REGION Network 2: Call: Diagnostic Profinet Devices
   // For diagnose the whole profinet devices of this PLC
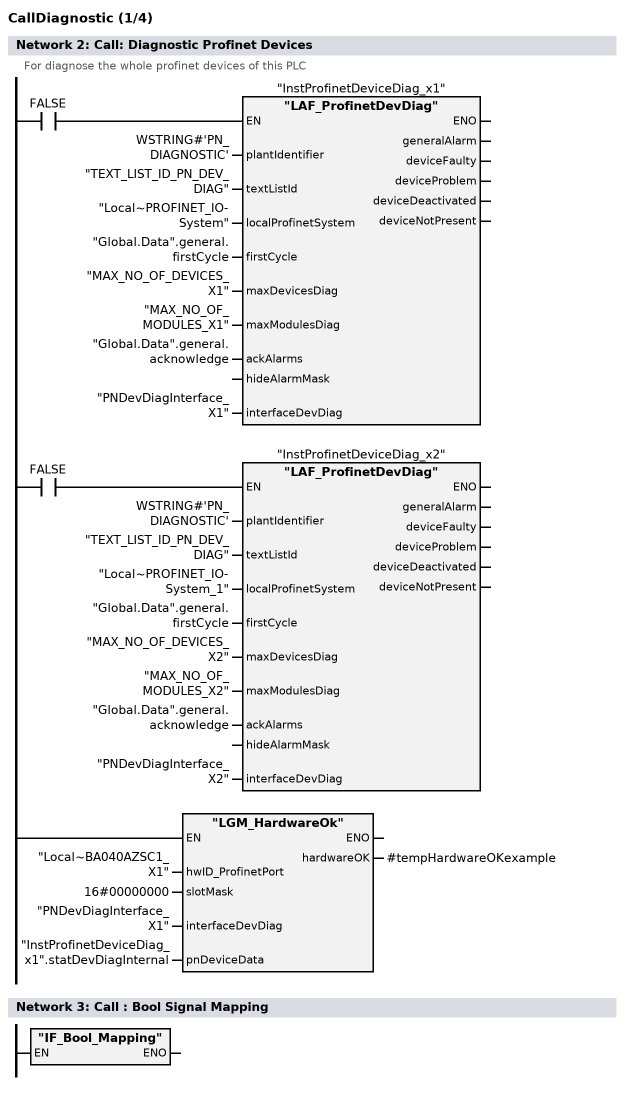
   RUNG wire#powerrail
      Contact( FALSE )
      "InstProfinetDeviceDiag_x1"(plantIdentifier := WSTRING#'PN_DIAGNOSTIC', textListId := "TEXT_LIST_ID_PN_DEV_DIAG", localProfinetSystem := "Local~PROFINET_IO-System", firstCycle := "Global.Data".general.firstCycle, maxDevicesDiag := "MAX_NO_OF_DEVICES_X1", maxModulesDiag := "MAX_NO_OF_MODULES_X1", ackAlarms := "Global.Data".general.acknowledge, hideAlarmMask :=, interfaceDevDiag := "PNDevDiagInterface_X1", generalAlarm =>, deviceFaulty =>, deviceProblem =>, deviceDeactivated =>, deviceNotPresent =>)
   END_RUNG
   RUNG wire#powerrail
      Contact( FALSE )
      "InstProfinetDeviceDiag_x2"(plantIdentifier := WSTRING#'PN_DIAGNOSTIC', textListId := "TEXT_LIST_ID_PN_DEV_DIAG", localProfinetSystem := "Local~PROFINET_IO-System_1", firstCycle := "Global.Data".general.firstCycle, maxDevicesDiag := "MAX_NO_OF_DEVICES_X2", maxModulesDiag := "MAX_NO_OF_MODULES_X2", ackAlarms := "Global.Data".general.acknowledge, hideAlarmMask :=, interfaceDevDiag := "PNDevDiagInterface_X2", generalAlarm =>, deviceFaulty =>, deviceProblem =>, deviceDeactivated =>, deviceNotPresent =>)
   END_RUNG
   RUNG wire#powerrail
      "LGM_HardwareOk"(hwID_ProfinetPort := "Local~BA040AZSC1_X1", slotMask := 16#00000000, interfaceDevDiag := "PNDevDiagInterface_X1", pnDeviceData := "InstProfinetDeviceDiag_x1".statDevDiagInternal, hardwareOK => #tempHardwareOKexample)
   END_RUNG
   // the same network as SCL:
   IF FALSE THEN
       "InstProfinetDeviceDiag_x1"(plantIdentifier := WSTRING#'PN_DIAGNOSTIC',   // "LAF_ProfinetDevDiag"
                               textListId := "TEXT_LIST_ID_PN_DEV_DIAG",
                               localProfinetSystem := "Local~PROFINET_IO-System",
                               firstCycle := "Global.Data".general.firstCycle,
                               maxDevicesDiag := "MAX_NO_OF_DEVICES_X1",
                               maxModulesDiag := "MAX_NO_OF_MODULES_X1",
                               ackAlarms := "Global.Data".general.acknowledge,
                               interfaceDevDiag := "PNDevDiagInterface_X1");
       "InstProfinetDeviceDiag_x2"(plantIdentifier := WSTRING#'PN_DIAGNOSTIC',   // "LAF_ProfinetDevDiag"
                               textListId := "TEXT_LIST_ID_PN_DEV_DIAG",
                               localProfinetSystem := "Local~PROFINET_IO-System_1",
                               firstCycle := "Global.Data".general.firstCycle,
                               maxDevicesDiag := "MAX_NO_OF_DEVICES_X2",
                               maxModulesDiag := "MAX_NO_OF_MODULES_X2",
                               ackAlarms := "Global.Data".general.acknowledge,
                               interfaceDevDiag := "PNDevDiagInterface_X2");
   END_IF;
   "LGM_HardwareOk"(hwID_ProfinetPort := "Local~BA040AZSC1_X1",
                    slotMask := 16#00000000,
                    interfaceDevDiag := "PNDevDiagInterface_X1",
                    pnDeviceData := "InstProfinetDeviceDiag_x1".statDevDiagInternal,
                    hardwareOK => #tempHardwareOKexample);
END_REGION

REGION Network 3: Call : Bool Signal Mapping
   RUNG wire#powerrail
      "IF_Bool_Mapping"()
   END_RUNG
   // the same network as SCL:
   "IF_Bool_Mapping"();
END_REGION

REGION Network 4: Call: Diagnostic Bool Interface Signals
   // Call the interface bool blocks to show boolean signals on the HMI
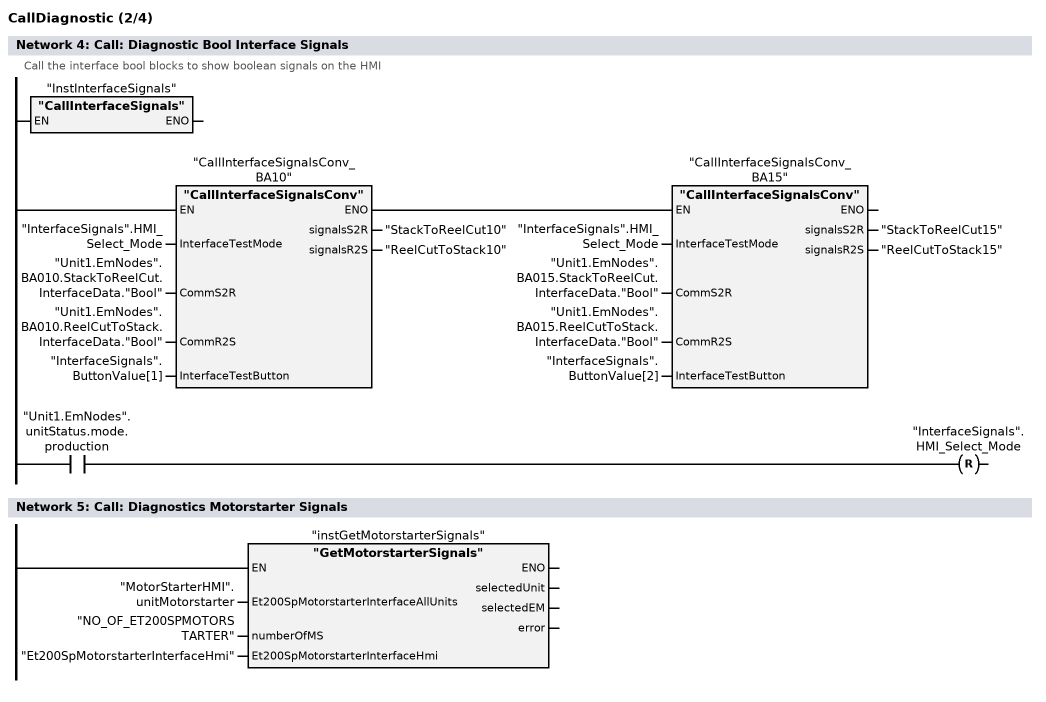
   RUNG wire#powerrail
      "InstInterfaceSignals"()
   END_RUNG
   RUNG wire#powerrail
      "CallInterfaceSignalsConv_BA10"(InterfaceTestMode := "InterfaceSignals".HMI_Select_Mode, CommS2R := "Unit1.EmNodes".BA010.StackToReelCut.InterfaceData."Bool", CommR2S := "Unit1.EmNodes".BA010.ReelCutToStack.InterfaceData."Bool", InterfaceTestButton := "InterfaceSignals".ButtonValue[1], signalsS2R => "StackToReelCut10", signalsR2S => "ReelCutToStack10")
      "CallInterfaceSignalsConv_BA15"(InterfaceTestMode := "InterfaceSignals".HMI_Select_Mode, CommS2R := "Unit1.EmNodes".BA015.StackToReelCut.InterfaceData."Bool", CommR2S := "Unit1.EmNodes".BA015.ReelCutToStack.InterfaceData."Bool", InterfaceTestButton := "InterfaceSignals".ButtonValue[2], signalsS2R => "StackToReelCut15", signalsR2S => "ReelCutToStack15")
   END_RUNG
   RUNG wire#powerrail
      Contact( "Unit1.EmNodes".unitStatus.mode.production )
      R_Coil( "InterfaceSignals".HMI_Select_Mode )
   END_RUNG
   // the same network as SCL:
   "InstInterfaceSignals"();   // "CallInterfaceSignals"
   "CallInterfaceSignalsConv_BA10"(InterfaceTestMode := "InterfaceSignals".HMI_Select_Mode,   // "CallInterfaceSignalsConv"
                           CommS2R := "Unit1.EmNodes".BA010.StackToReelCut.InterfaceData."Bool",
                           CommR2S := "Unit1.EmNodes".BA010.ReelCutToStack.InterfaceData."Bool",
                           InterfaceTestButton := "InterfaceSignals".ButtonValue[1],
                           signalsS2R => "StackToReelCut10",
                           signalsR2S => "ReelCutToStack10",
                           ENO => #_w1);
   IF #_w1 THEN
       "CallInterfaceSignalsConv_BA15"(InterfaceTestMode := "InterfaceSignals".HMI_Select_Mode,   // "CallInterfaceSignalsConv"
                               CommS2R := "Unit1.EmNodes".BA015.StackToReelCut.InterfaceData."Bool",
                               CommR2S := "Unit1.EmNodes".BA015.ReelCutToStack.InterfaceData."Bool",
                               InterfaceTestButton := "InterfaceSignals".ButtonValue[2],
                               signalsS2R => "StackToReelCut15",
                               signalsR2S => "ReelCutToStack15");
   END_IF;
   IF "Unit1.EmNodes".unitStatus.mode.production THEN "InterfaceSignals".HMI_Select_Mode := FALSE; END_IF;
END_REGION

REGION Network 5: Call: Diagnostics Motorstarter Signals
   RUNG wire#powerrail
      "instGetMotorstarterSignals"(Et200SpMotorstarterInterfaceAllUnits := "MotorStarterHMI".unitMotorstarter, numberOfMS := "NO_OF_ET200SPMOTORSTARTER", Et200SpMotorstarterInterfaceHmi := "Et200SpMotorstarterInterfaceHmi", selectedUnit =>, selectedEM =>, error =>)
   END_RUNG
   // the same network as SCL:
   "instGetMotorstarterSignals"(Et200SpMotorstarterInterfaceAllUnits := "MotorStarterHMI".unitMotorstarter,   // "GetMotorstarterSignals"
                           numberOfMS := "NO_OF_ET200SPMOTORSTARTER",
                           Et200SpMotorstarterInterfaceHmi := "Et200SpMotorstarterInterfaceHmi");
END_REGION

REGION Network 6: Call: Diagnostics Drives
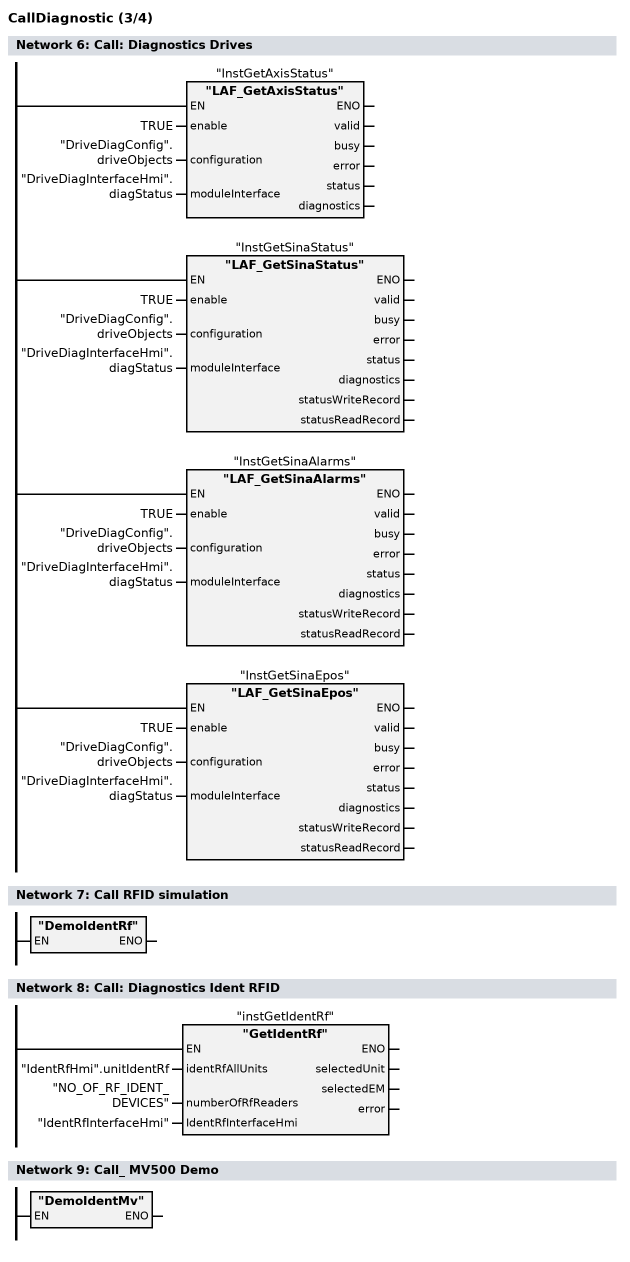
   RUNG wire#powerrail
      "InstGetAxisStatus"(enable := TRUE, configuration := "DriveDiagConfig".driveObjects, moduleInterface := "DriveDiagInterfaceHmi".diagStatus, valid =>, busy =>, error =>, status =>, diagnostics =>)
   END_RUNG
   RUNG wire#powerrail
      "InstGetSinaStatus"(enable := TRUE, configuration := "DriveDiagConfig".driveObjects, moduleInterface := "DriveDiagInterfaceHmi".diagStatus, valid =>, busy =>, error =>, status =>, diagnostics =>, statusWriteRecord =>, statusReadRecord =>)
   END_RUNG
   RUNG wire#powerrail
      "InstGetSinaAlarms"(enable := TRUE, configuration := "DriveDiagConfig".driveObjects, moduleInterface := "DriveDiagInterfaceHmi".diagStatus, valid =>, busy =>, error =>, status =>, diagnostics =>, statusWriteRecord =>, statusReadRecord =>)
   END_RUNG
   RUNG wire#powerrail
      "InstGetSinaEpos"(enable := TRUE, configuration := "DriveDiagConfig".driveObjects, moduleInterface := "DriveDiagInterfaceHmi".diagStatus, valid =>, busy =>, error =>, status =>, diagnostics =>, statusWriteRecord =>, statusReadRecord =>)
   END_RUNG
   // the same network as SCL:
   "InstGetAxisStatus"(enable := TRUE,   // "LAF_GetAxisStatus"
                       configuration := "DriveDiagConfig".driveObjects,
                       moduleInterface := "DriveDiagInterfaceHmi".diagStatus);
   "InstGetSinaStatus"(enable := TRUE,   // "LAF_GetSinaStatus"
                       configuration := "DriveDiagConfig".driveObjects,
                       moduleInterface := "DriveDiagInterfaceHmi".diagStatus);
   "InstGetSinaAlarms"(enable := TRUE,   // "LAF_GetSinaAlarms"
                       configuration := "DriveDiagConfig".driveObjects,
                       moduleInterface := "DriveDiagInterfaceHmi".diagStatus);
   "InstGetSinaEpos"(enable := TRUE,   // "LAF_GetSinaEpos"
                     configuration := "DriveDiagConfig".driveObjects,
                     moduleInterface := "DriveDiagInterfaceHmi".diagStatus);
END_REGION

REGION Network 7: Call RFID simulation
   RUNG wire#powerrail
      "DemoIdentRf"()
   END_RUNG
   // the same network as SCL:
   "DemoIdentRf"();
END_REGION

REGION Network 8: Call: Diagnostics Ident RFID
   RUNG wire#powerrail
      "instGetIdentRf"(identRfAllUnits := "IdentRfHmi".unitIdentRf, numberOfRfReaders := "NO_OF_RF_IDENT_DEVICES", IdentRfInterfaceHmi := "IdentRfInterfaceHmi", selectedUnit =>, selectedEM =>, error =>)
   END_RUNG
   // the same network as SCL:
   "instGetIdentRf"(identRfAllUnits := "IdentRfHmi".unitIdentRf,   // "GetIdentRf"
                    numberOfRfReaders := "NO_OF_RF_IDENT_DEVICES",
                    IdentRfInterfaceHmi := "IdentRfInterfaceHmi");
END_REGION

REGION Network 9: Call_ MV500 Demo
   RUNG wire#powerrail
      "DemoIdentMv"()
   END_RUNG
   // the same network as SCL:
   "DemoIdentMv"();
END_REGION

REGION Network 10: Call: Diagnosticsa Ident MV
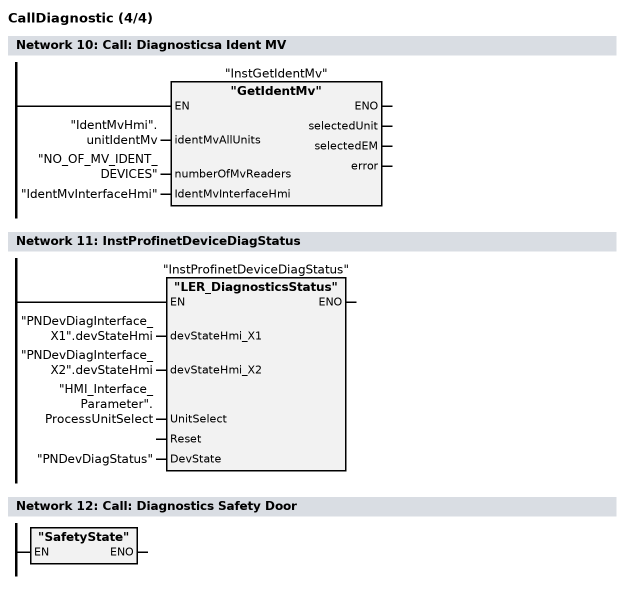
   RUNG wire#powerrail
      "InstGetIdentMv"(identMvAllUnits := "IdentMvHmi".unitIdentMv, numberOfMvReaders := "NO_OF_MV_IDENT_DEVICES", IdentMvInterfaceHmi := "IdentMvInterfaceHmi", selectedUnit =>, selectedEM =>, error =>)
   END_RUNG
   // the same network as SCL:
   "InstGetIdentMv"(identMvAllUnits := "IdentMvHmi".unitIdentMv,   // "GetIdentMv"
                    numberOfMvReaders := "NO_OF_MV_IDENT_DEVICES",
                    IdentMvInterfaceHmi := "IdentMvInterfaceHmi");
END_REGION

REGION Network 11: InstProfinetDeviceDiagStatus
   RUNG wire#powerrail
      "InstProfinetDeviceDiagStatus"(devStateHmi_X1 := "PNDevDiagInterface_X1".devStateHmi, devStateHmi_X2 := "PNDevDiagInterface_X2".devStateHmi, UnitSelect := "HMI_Interface_Parameter".ProcessUnitSelect, Reset :=, DevState := "PNDevDiagStatus")
   END_RUNG
   // the same network as SCL:
   "InstProfinetDeviceDiagStatus"(devStateHmi_X1 := "PNDevDiagInterface_X1".devStateHmi,   // "LER_DiagnosticsStatus"
                           devStateHmi_X2 := "PNDevDiagInterface_X2".devStateHmi,
                           UnitSelect := "HMI_Interface_Parameter".ProcessUnitSelect,
                           DevState := "PNDevDiagStatus");
END_REGION

REGION Network 12: Call: Diagnostics Safety Door
   RUNG wire#powerrail
      "SafetyState"()
   END_RUNG
   // the same network as SCL:
   "SafetyState"();
END_REGION
END_FUNCTION

FUNCTION "IF_Bool_Mapping" : Void
{ S7_Optimized_Access := 'TRUE' ; Published := 'FALSE' }
VERSION : 0.1

BEGIN
	// IO Mapping 25.12.10
	REGION BK
	    REGION BK01
	        "BK01"."X10-1.BTM DIRECTION CHECK SENSOR" := "BA040AZSBK01.00";
	        //"BK01"."X11-1.SPARE" := "BA030AZSBK01.I01";
	        //"BK01"."X12-1.SPARE" := "BA030AZSBK01.I02";
	        "BK01"."X13-1.COMPENSATOR #1 LIMIT SENSOR(-)" := "Sensor".EM3[0];
	        "BK01"."X14-1.COMPENSATOR #1 LIMIT SENSOR(+)" := "Sensor".EM3[1];
	        //"BK01"."X15-1.SPARE" := "BA030AZSBK01.I05";
	        //"BK01"."X16-1.SPARE" := "BA030AZSBK01.I06";
	        "BK01"."X17-1.SAFETY PIN IDLE POSITION" := "BA040AZSBK01.07";
	        "BK01"."X10-2.TOP DIRECTION CHECK SENSOR" := "BA040AZSBK01.10";
	        //"BK01"."X11-2.SPARE" := "BA030AZSBK01.I09";
	        //"BK01"."X12-2.SPARE" := "BA030AZSBK01.I10";
	        "BK01"."X13-2.COMPENSATOR #1 HOME SENSOR" := "Sensor".EM3[2];
	        //"BK01"."X14-2.SPARE" := "BA030AZSBK01.I12";
	        //"BK01"."X15-2.SPARE" := "BA030AZSBK01.I13";
	        //"BK01"."X16-2.SPARE" := "BA030AZSBK01.I14";
	        //"BK01"."X17-2.SPARE" := "BA030AZSBK01.I15";
	    END_REGION
	    REGION BK02
	        "BK02"."X10-1.SUCTION PAD TOP DOWN" := "BA040AZSBK02.00";
	        "BK02"."X11-1.SUCTION PAD BTM DOWN" := "BA040AZSBK02.01";
	        "BK02"."X12-1.CUTTER DOWN" := "BA040AZSBK02.02";
	        "BK02"."X13-1.TAPE TOP DOWN" := "BA040AZSBK02.03";
	        "BK02"."X14-1.TAPE BTM DOWN" := "BA040AZSBK02.04";
	        "BK02"."X15-1.SPLICE HEAD ROTATE TOP BACKWARD" := "BA040AZSBK02.05";
	        "BK02"."X16-1.SPLICE HEAD ROTATE BTM BACKWARD" := "BA040AZSBK02.06";
	        //"BK02"."X17-1.SPARE" := "BA030AZSBK02.I07";
	        "BK02"."X10-2.SUCTION PAD TOP UP" := "BA040AZSBK02.10";
	        "BK02"."X11-2.SUCTION PAD BTM UP" := "BA040AZSBK02.11";
	        "BK02"."X12-2.CUTTER UP" := "BA040AZSBK02.12";
	        "BK02"."X13-2.TAPE TOP UP" := "BA040AZSBK02.13";
	        "BK02"."X14-2.TAPE BTM UP" := "BA040AZSBK02.14";
	        "BK02"."X15-2.SPLICE HEAD ROTATE TOP FORWARD" := "BA040AZSBK02.15";
	        "BK02"."X16-2.SPLICE HEAD ROTATE BTM FORWARD" := "BA040AZSBK02.16";
	        //"BK02"."X17-2.SPARE" := "BA030AZSBK02.I15";
	    END_REGION
	    REGION BK03
	        "BK03"."X10-1.SUCTION PAD TOP LEFT PRESSURE SWITCH" := "BA040AZSBK03.00";
	        "BK03"."X10-2.SUCTION PAD TOP RIGHT PRESSURE SWITCH" := "BA040AZSBK03.01";
	        "BK03"."X12-1.SUCTION PAD BTM LEFT PRESSURE SWITCH" := "BA040AZSBK03.02";
	        "BK03"."X12-2.SUCTION PAD BTM RIGHT PRESSURE SWITCH" := "BA040AZSBK03.03";
	        "BK03"."X14-1.SUCTION PAD TOP TAPE PRESSURE SWITCH" := "BA040AZSBK03.04";
	        "BK03"."X14-2.SUCTION PAD BTM TAPE PRESSURE SWITCH" := "BA040AZSBK03.05";
	        "BK03"."X14-2.SUCTION PAD BTM TAPE PRESSURE SWITCH" := "BA040AZSBK03.06";
	        //"BK03"."X16-2.SPARE" := "BA030AZSBK03.I07";
	    END_REGION
	    REGION BK04
	        "BK04"."X10-1.CATHODE MAIN P&P1 LIMITS SENSOR(-)" := "Sensor".EM5[18];
	        "BK04"."X11-1.CATHODE MAIN P&P1 LIMITS SENSOR(+)" := "Sensor".EM5[19];
	        "BK04"."X12-1.CATHODE MAIN P&P2 LIMITS SENSOR(-)" := "Sensor".EM5[21];
	        "BK04"."X13-1.CATHODE MAIN P&P2 LIMITS SENSOR(+)" := "Sensor".EM5[22];
	        "BK04"."X14-1.ANODE MAIN P&P2 LIMITS SENSOR(-)" := "Sensor".EM4[0];
	        "BK04"."X15-1.ANODE MAIN P&P2 LIMITS SENSOR(+)" := "Sensor".EM4[1];
	        "BK04"."X16-1.ANODE MAIN P&P1 LIMITS SENSOR(-)" := "Sensor".EM4[21];
	        "BK04"."X17-1.ANODE MAIN P&P1 LIMITS SENSOR(+)" := "Sensor".EM4[22];
	        "BK04"."X10-2.CATHODE MAIN P&P1 LIMITS SENSOR HOME" := "Sensor".EM5[20];
	        //"BK04"."X11-2.SPARE" := "BA030AZSBK04.I09";
	        "BK04"."X12-2.CATHODE MAIN P&P2 LIMITS SENSOR HOME" := "Sensor".EM5[23];
	        //"BK04"."X13-2.SPARE" := "BA030AZSBK04.I11";
	        "BK04"."X14-2.ANODE MAIN P&P2 LIMITS SENSOR HOME" := "Sensor".EM4[2];
	        //"BK04"."X15-2.SPARE" := "BA030AZSBK04.I13";
	        "BK04"."X16-2.ANODE MAIN P&P1 LIMITS SENSOR HOME" := "Sensor".EM4[23];
	        //"BK04"."X17-2.SPARE" := "BA030AZSBK04.I15";
	    END_REGION
	    REGION BK05
	        "BK05"."X10-1.ANODE MAIN P&P1 Z-AXIS LIMIT SENSOR(-)" := "Sensor".EM4[3];
	        "BK05"."X11-1.ANODE MAIN P&P1 Z-AXIS LIMIT SENSOR(+)" := "Sensor".EM4[4];
	        "BK05"."X12-1.ANODE MAIN P&P1 Y-AXIS LIMIT SENSOR(-)" := "Sensor".EM4[5];
	        "BK05"."X13-1.ANODE MAIN P&P1 Y-AXIS LIMIT SENSOR(+)" := "Sensor".EM4[6];
	        //"BK05"."X14-1.SPARE" := "BA030AZSBK05.I04";
	        "BK05"."X15-1.ANODE MAIN P&P1 DETECT SENSOR" := "BA040AZSBK05.05";
	        "BK05"."X16-1.ANODE MAIN P&P1 ROTARY CCW" := "BA040AZSBK05.06";
	        "BK05"."X17-1.ANODE MAIN P&P1 PRESSURE SWITCH" := "BA040AZSBK05.07";
	        "BK05"."X10-2.ANODE MAIN P&P1 Z-AXIS HOME SENSOR" := "Sensor".EM4[7];
	        //"BK05"."X11-2.SPARE" := "BA030AZSBK05.I09";
	        "BK05"."X12-2.ANODE MAIN P&P1 Y-AXIS HOME SENSOR" := "Sensor".EM4[8];
	        //"BK05"."X13-2.SPARE" := "BA030AZSBK05.I11";
	        //"BK05"."X14-2.SPARE" := "BA030AZSBK05.I12";
	        //"BK05"."X15-2.SPARE" := "BA030AZSBK05.I13";
	        "BK05"."X16-2.ANODE MAIN P&P1 ROTARY CW" := "BA040AZSBK05.16";
	        //"BK05"."X17-2.SPARE" := "BA030AZSBK05.I15";
	    END_REGION BK06
	        "BK06"."X10-1.ANODE MAIN P&P2 Z-AXIS LIMIT SENSOR(-)" := "Sensor".EM4[9];
	        "BK06"."X10-2.ANODE MAIN P&P2 Z-AXIS HOME SENSOR" := "Sensor".EM4[10];
	        "BK06"."X12-1.ANODE MAIN P&P2 Z-AXIS LIMIT SENSOR(+)" := "Sensor".EM4[11];
	        "BK06"."X12-2.ANODE MAIN P&P2 DETECT SENSOR" := "BA040AZSBK06.03";
	        "BK06"."X14-1.ANODE MAIN P&P2 PRESSURE SWITCH" := "BA040AZSBK06.04";
	        //"BK06"."X14-2.SPARE" := "BA030AZSBK06.I05";
	        //"BK06"."X16-1.SPARE" := "BA030AZSBK06.I06";
	        //"BK06"."X16-2.SPARE" := "BA030AZSBK06.I07";
	    REGION BK07
	        "BK07"."X10-1.CATHODE MAIN P&P1 Z-AXIS LIMIT SENSOR(-)" := "Sensor".EM5[0];
	        "BK07"."X11-1.CATHODE MAIN P&P1 Z-AXIS LIMIT SENSOR(+)" := "Sensor".EM5[1];
	        "BK07"."X12-1.CATHODE MAIN P&P1 Y-AXIS LIMIT SENSOR(-)" := "Sensor".EM5[2];
	        "BK07"."X13-1.CATHODE MAIN P&P1 Y-AXIS LIMIT SENSOR(+)" := "Sensor".EM5[3];
	        //"BK07"."X14-1.SPARE" := "BA030AZSBK07.I04";
	        "BK07"."X15-1.CATHODE MAIN P&P1 DETECT SENSOR" := "BA040AZSBK07.05";
	        "BK07"."X16-1.CATHODE MAIN P&P1 ROTARY CCW" := "BA040AZSBK07.06";
	        "BK07"."X17-1.CATHODE MAIN P&P1 PRESSURE SWITCH" := "BA040AZSBK07.07";
	        "BK07"."X10-2.CATHODE MAIN P&P1 Z-AXIS HOME SENSOR" := "Sensor".EM5[4];
	        "BK07"."X12-2.CATHODE MAIN P&P1 Y-AXIS HOME SENSOR" := "Sensor".EM5[5];
	        //"BK07"."X14-2.SPARE" := "BA030AZSBK07.I12";
	        //"BK07"."X16-2.CATHODE MAIN P&P1 ROTARY CW" := "BA030AZSBK07.I.15";
	    END_REGION
	    REGION BK08
	        "BK08"."X10-1.CATHODE MAIN P&P2 Z-AXIS LIMIT SENSOR(-)" := "Sensor".EM5[6];
	        "BK08"."X12-1.CATHODE MAIN P&P2 Z-AXIS LIMIT SENSOR(+)" := "Sensor".EM5[8];
	        "BK08"."X14-1.CATHODE MAIN P&P2 PRESSURE SWITCH" := "BA040AZSBK08.04";
	        "BK08"."X10-2.CATHODE MAIN P&P2 Z-AXIS HOME SENSOR" := "Sensor".EM5[7];
	        "BK08"."X12-2.CATHODE MAIN P&P2 DETECT SENSOR" := "BA040AZSBK08.03";
	    END_REGION
	    REGION BK09
	        "BK09"."X10-1.ANODE ALIGN TABLE Y2-AXIS LIMIT SENSOR(-)" := "Sensor".EM4[12];
	        "BK09"."X11-1.ANODE ALIGN TABLE Y2-AXIS LIMIT SENSOR(+)" := "Sensor".EM4[13];
	        "BK09"."X12-1.ANODE ALIGN TABLE X-AXIS LIMIT SENSOR(-)" := "Sensor".EM4[14];
	        "BK09"."X13-1.ANODE ALIGN TABLE X-AXIS LIMIT SENSOR(+)" := "Sensor".EM4[15];
	        "BK09"."X14-1.ANODE ALIGN TABLE Y1-AXIS LIMIT SENSOR(-)" := "Sensor".EM4[16];
	        "BK09"."X15-1.ANODE ALIGN TABLE Y1-AXIS LIMIT SENSOR(+)" := "Sensor".EM4[17];
	        "BK09"."X16-1.ANODE ALIGN TABLE ELECTRODE DETECT SENSOR" := "BA040AZSBK09.06";
	        "BK09"."X17-1.ANODE ALIGN TABLE PRESSURE SWITCH" := "BA040AZSBK09.07";
	        "BK09"."X10-2.ANODE ALIGN TABLE Y2-AXIS HOME SENSOR" := "Sensor".EM4[18];
	        "BK09"."X12-2.ANODE ALIGN TABLE X-AXIS HOME SENSOR" := "Sensor".EM4[19];
	        "BK09"."X14-2.ANODE ALIGN TABLE Y1-AXIS HOME SENSOR" := "Sensor".EM4[20];
	    END_REGION
	    REGION BK10
	        "BK10"."X10-1.ANODE FIX FRONT BACKWARD" := "BA040AZSBK10.00";
	        "BK10"."X11-1.SEPA CLAMP SAFETY PIN DETECT SENSOR" := "BA040AZSBK10.01";
	        "BK10"."X12-1.ANODE FIX REAR BACKWARD" := "BA040AZSBK10.02";
	        "BK10"."X13-1.SEPA CLAMP PRESSURE SWITCH" := "BA040AZSBK10.03";
	        "BK10"."X14-1.FIX ANODE DETECT SENSOR" := "BA040AZSBK10.04";
	        "BK10"."X10-2.ANODE FIX FRONT FORWARD" := "BA040AZSBK10.10";
	        "BK10"."X11-2.SEPA GRIPPER SAFETY PIN DETECT SENSOR" := "BA040AZSBK10.11";
	        "BK10"."X12-2.ANODE FIX REAR FORWARD" := "BA040AZSBK10.12";
	    END_REGION
	    REGION BK11
	        "BK11"."X10-1.ANODE NG BOX FULL SENSOR" := "BA040AZSBK11.00";
	        //"BK11"."X10-2.SPARE" := "BA030AZSBK11.I01";
	        "BK11"."X12-1.ANODE NG BOX LIFT DOWN" := "BA040AZSBK11.02";
	        "BK11"."X12-2.ANODE NG BOX LIFT UP" := "BA040AZSBK11.03";
	        "BK11"."X14-1.ANODE NG BOX LOCK DOWN" := "BA040AZSBK11.04";
	        "BK11"."X14-2.ANODE NG BOX LOCK UP" := "BA040AZSBK11.05";
	        "BK11"."X16-1.ANODE NG BOX NG BOX DETECT SENSOR" := "BA040AZSBK11.06";
	    END_REGION
	    REGION BK12
	        "BK12"."X10-1.ANODE NG P&P 1st BACKWARD" := "BA040AZSBK12.00";
	        "BK12"."X12-1.ANODE NG P&P 2nd BACKWARD" := "BA040AZSBK12.02";
	        "BK12"."X14-1.ANODE NG P&P UP" := "BA040AZSBK12.04";
	        "BK12"."X16-1.ANODE NG P&P VACUUM PRESSURE SWITCH" := "BA040AZSBK12.06";
	        "BK12"."X10-2.ANODE NG P&P 1st FORWARD" := "BA040AZSBK12.10";
	        "BK12"."X12-2.ANODE NG P&P 2nd FORWARD" := "BA040AZSBK12.12";
	        "BK12"."X14-2.ANODE NG P&P DOWN" := "BA040AZSBK12.14";
	        "BK12"."X16-2.ANODE NG P&P ELECTRODE DETECT SENSOR" := "BA040AZSBK12.16";
	    END_REGION
	    REGION BK13
	        "BK13"."X10-1.CATHODE ALIGN TABLE Y1-AXIS LIMIT SENSOR(-)" := "Sensor".EM5[10];
	        "BK13"."X11-1.CATHODE ALIGN TABLE Y1-AXIS LIMIT SENSOR(+)" := "Sensor".EM5[9];
	        "BK13"."X12-1.CATHODE ALIGN TABLE X-AXIS LIMIT SENSOR(-)" := "Sensor".EM5[11];
	        "BK13"."X13-1.CATHODE ALIGN TABLE X-AXIS LIMIT SENSOR(+)" := "Sensor".EM5[12];
	        "BK13"."X14-1.CATHODE ALIGN TABLE Y2-AXIS LIMIT SENSOR(-)" := "Sensor".EM5[13];
	        "BK13"."X15-1.CATHODE ALIGN TABLE Y2-AXIS LIMIT SENSOR(+)" := "Sensor".EM5[14];
	        "BK13"."X16-1.CATHODE ALIGN TABLE ELECTRODE DETECT SENSOR" := "BA040AZSBK13.06";
	        "BK13"."X17-1.CATHODE ALIGN TABLE PRESSURE SWITCH" := "BA040AZSBK13.07";
	        "BK13"."X10-2.CATHODE ALIGN TABLE Y1-AXIS HOME SENSOR" := "Sensor".EM5[17];
	        "BK13"."X12-2.CATHODE ALIGN TABLE X-AXIS HOME SENSOR" := "Sensor".EM5[15];
	    END_REGION
	    REGION BK14
	        "BK14"."X10-1.FIX CATHODE FRONT BACKWARD" := "BA040AZSBK14.00";
	        "BK14"."X11-1.STACK TABLE OUT REAR Z-AXIS LIMIT SENSOR(-)" := "Sensor".EM6[36];
	        "BK14"."X12-1.FIX CATHODE REAR BACKWARD" := "BA040AZSBK14.02";
	        "BK14"."X13-1.STACK TABLE OUT REAR Z-AXIS LIMIT SENSOR(+)" := "Sensor".EM6[37];
	        "BK14"."X14-1.FIX CATHODE DETECT SENSOR" := "BA040AZSBK14.04";
	        "BK14"."X10-2.FIX CATHODE FRONT FORWARD" := "BA040AZSBK14.10";
	        "BK14"."X11-2.STACK TABLE OUT REAR Z-AXIS HOME SENSOR" := "Sensor".EM6[38];
	        "BK14"."X12-2.FIX CATHODE REAR FORWARD" := "BA040AZSBK14.12";
	    END_REGION
	    REGION BK15
	        "BK15"."X10-1.CATHODE NG BOX FULL SENSOR" := "BA040AZSBK15.00";
	        "BK15"."X10-2.CATHODE NG BOX NG BOX DETECT SENSOR" := "BA040AZSBK15.01";
	        "BK15"."X12-1.CATHODE NG BOX LIFT DOWN" := "BA040AZSBK15.02";
	        "BK15"."X12-2.CATHODE NG BOX LIFT UP" := "BA040AZSBK15.03";
	        "BK15"."X14-1.CATHODE NG BOX LOCK DOWN" := "BA040AZSBK15.04";
	        "BK15"."X14-2.CATHODE NG BOX LOCK UP" := "BA040AZSBK15.05";
	    END_REGION
	    REGION BK16
	        "BK16"."X10-1.CATHODE NG P&P 1st BACKWARD" := "BA040AZSBK16.00";
	        "BK16"."X12-1.CATHODE NG P&P 2nd BACKWARD" := "BA040AZSBK16.02";
	        "BK16"."X14-1.CATHODE NG P&P DOWN" := "BA040AZSBK16.04";
	        "BK16"."X16-1.CATHODE NG P&P VACUUM PRESSURE SWITCH" := "BA040AZSBK16.06";
	        "BK16"."X10-2.CATHODE NG P&P 1st FORWARD" := "BA040AZSBK16.10";
	        "BK16"."X12-2.CATHODE NG P&P 2nd FORWARD" := "BA040AZSBK16.12";
	        "BK16"."X14-2.CATHODE NG P&P UP" := "BA040AZSBK16.14";
	        "BK16"."X16-2.CATHODE NG P&P ELECTRODE DETECT SENSOR" := "BA040AZSBK16.16";
	    END_REGION ;
	    REGION BK17
	        "BK17"."X10-1.FINAL ROLLER FRONT LIMIT SENSOR(-)" := "Sensor".EM6[0];
	        "BK17"."X10-2.FINAL ROLLER FRONT HOME SENSOR" := "Sensor".EM6[1];
	        "BK17"."X12-1.FINAL ROLLER FRONT LIMIT SENSOR(+)" := "Sensor".EM6[2];
	        "BK17"."X14-1.FINAL ROLLER REAR LIMIT SENSOR(-)" := "Sensor".EM6[3];
	        "BK17"."X14-2.FINAL ROLLER REAR HOME SENSOR" := "Sensor".EM6[4];
	        "BK17"."X16-1.FINAL ROLLER REAR LIMIT SENSOR(+)" := "Sensor".EM6[5];
	    END_REGION
	    REGION BK18
	        "BK18"."X10-1.ANODE MANDREL REAR Y AXIS LIMIT SENSOR(-)" := "Sensor".EM6[6];
	        "BK18"."X11-1.ANODE MANDREL REAR Y AXIS LIMIT SENSOR(+)" := "Sensor".EM6[7];
	        "BK18"."X12-1.ANODE MANDREL REAR Z AXIS LIMIT SENSOR(-)" := "Sensor".EM6[8];
	        "BK18"."X13-1.ANODE MANDREL REAR Z AXIS LIMIT SENSOR(+)" := "Sensor".EM6[9];
	        "BK18"."X14-1.ANODE MANDREL FRONT Y AXIS LIMIT SENSOR(-)" := "Sensor".EM6[10];
	        "BK18"."X15-1.ANODE MANDREL FRONT Y AXIS LIMIT SENSOR(+)" := "Sensor".EM6[11];
	        "BK18"."X16-1.ANODE MANDREL FRONT Z AXIS LIMIT SENSOR(-)" := "Sensor".EM6[12];
	        "BK18"."X17-1.ANODE MANDREL FRONT Z AXIS LIMIT SENSOR(+)" := "Sensor".EM6[13];
	        "BK18"."X10-2.ANODE MANDREL REAR Y AXIS HOME SENSOR" := "Sensor".EM6[14];
	        "BK18"."X12-2.ANODE MANDREL REAR Z AXIS HOME SENSOR" := "Sensor".EM6[15];
	        "BK18"."X14-2.ANODE MANDREL FRONT Y AXIS HOME SENSOR" := "Sensor".EM6[16];
	        "BK18"."X16-2.ANODE MANDREL FRONT Z AXIS HOME SENSOR" := "Sensor".EM6[17];
	    END_REGION
	    REGION BK19
	        "BK19"."X10-1.CATHODE MANDREL REAR Y AXIS LIMIT SENSOR(-)" := "Sensor".EM6[18];
	        "BK19"."X11-1.CATHODE MANDREL REAR Y AXIS LIMIT SENSOR(+)" := "Sensor".EM6[19];
	        "BK19"."X12-1.CATHODE MANDREL REAR Z AXIS LIMIT SENSOR(-)" := "Sensor".EM6[20];
	        "BK19"."X13-1.CATHODE MANDREL REAR Z AXIS LIMIT SENSOR(+)" := "Sensor".EM6[21];
	        "BK19"."X14-1.CATHODE MANDREL FRONT Y AXIS LIMIT SENSOR(-)" := "Sensor".EM6[22];
	        "BK19"."X15-1.CATHODE MANDREL FRONT Y AXIS LIMIT SENSOR(+)" := "Sensor".EM6[23];
	        "BK19"."X16-1.CATHODE MANDREL FRONT Z AXIS LIMIT SENSOR(-)" := "Sensor".EM6[24];
	        "BK19"."X17-1.CATHODE MANDREL FRONT Z AXIS LIMIT SENSOR(+)" := "Sensor".EM6[25];
	        "BK19"."X10-2.CATHODE MANDREL REAR Y AXIS HOME SENSOR" := "Sensor".EM6[26];
	        "BK19"."X12-2.CATHODE MANDREL REAR Z AXIS HOME SENSOR" := "Sensor".EM6[27];
	        "BK19"."X14-2.CATHODE MANDREL FRONT Y AXIS HOME SENSOR" := "Sensor".EM6[28];
	        "BK19"."X16-2.CATHODE MANDREL FRONT Z AXIS HOME SENSOR" := "Sensor".EM6[29];
	    END_REGION
	    REGION BK20
	        "BK20"."X10-1.STACK TABLE Z-AXIS LIMIT SENSOR(-)" := "Sensor".EM6[30];
	        "BK20"."X11-1.STACK TABLE Z-AXIS LIMIT SENSOR(+)" := "Sensor".EM6[31];
	        "BK20"."X12-1.STACK TABLE GAP PAD DOWN" := "BA040AZSBK20.02";
	        "BK20"."X13-1.STACK TABLE GAP PAD UP" := "BA040AZSBK20.03";
	        "BK20"."X14-1.STACK TABLE OUT FRONT Z-AXIS LIMIT SENSOR(-)" := "Sensor".EM6[32];
	        "BK20"."X15-1.STACK TABLE OUT FRONT Z-AXIS LIMIT SENSOR(+)" := "Sensor".EM6[33];
	        "BK20"."X16-1.STACK TABLE VACUUM PRESSURE SWITCH" := "BA040AZSBK20.06";
	        "BK20"."X10-2.STACK TABLE Z-AXIS HOME SENSOR" := "Sensor".EM6[34];
	        "BK20"."X14-2.STACK TABLE OUT FRONT Z-AXIS HOME SENSOR" := "Sensor".EM6[35];
	        "BK20"."X16-2.STACK TABLE ELECTRODE DETECT SENSOR" := "BA040AZSBK20.16";
	    END_REGION
	    REGION BK21
	        "BK21"."X10-1.SEPA CLAMP&CUTTER X-AXIS LIMIT SENSOR(-)" := "Sensor".EM7[0];
	        "BK21"."X10-2.SEPA CLAMP&CUTTER X-AXIS HOME SENSOR" := "Sensor".EM7[1];
	        "BK21"."X12-1.SEPA CLAMP&CUTTER X-AXIS LIMIT SENSOR(+)" := "Sensor".EM7[2];
	        "BK21"."X14-1.SEPA GRIPPER X-AXIS LIMIT SENSOR(-)" := "Sensor".EM7[3];
	        "BK21"."X14-2.SEPA GRIPPER X-AXIS HOME SENSOR" := "Sensor".EM7[4];
	        "BK21"."X16-1.SEPA GRIPPER X-AXIS LIMIT SENSOR(+)" := "Sensor".EM7[5];
	    END_REGION
	    REGION BK22
	        "BK22"."X10-1.SEPA GRIPPER CLAMP OPEN" := "BA040AZSBK22.00";
	        "BK22"."X12-1.SEPA GRIPPER CLAMP DETECT SENSOR" := "BA040AZSBK22.02";
	        "BK22"."X13-1.SEPA GRIPPER BACKWARD" := "BA040AZSBK22.03";
	        "BK22"."X14-1.SEPA GRIPPER C-AXIS LIMIT SENSOR(-)" := "Sensor".EM7[20];
	        "BK22"."X15-1.SEPA GRIPPER C-AXIS LIMIT SENSOR(+)" := "Sensor".EM7[6];
	        "BK22"."X16-1.SEPA GRIPPER Z-AXIS LIMIT SENSOR(-)" := "Sensor".EM7[7];
	        "BK22"."X17-1.SEPA GRIPPER Z-AXIS LIMIT SENSOR(+)" := "Sensor".EM7[8];
	        "BK22"."X10-2.SEPA GRIPPER CLAMP CLOSE" := "BA040AZSBK22.10";
	        "BK22"."X13-2.SEPA GRIPPER FORWARD" := "BA040AZSBK22.13";
	        "BK22"."X14-2.SEPA GRIPPER C-AXIS HOME SENSOR" := "Sensor".EM7[24];
	        "BK22"."X16-2.SEPA GRIPPER Z-AXIS HOME SENSOR" := "Sensor".EM7[9];
	    END_REGION
	    REGION BK23    
	        "BK23"."X10-1.SEPA CLAMP&CUTTER Z-AXIS LIMIT SENSOR(-)" := "Sensor".EM7[11];
	        "BK23"."X11-1.SEPA CLAMP&CUTTER Z-AXIS LIMIT SENSOR(+)" := "Sensor".EM7[12];
	        "BK23"."X12-1.SEPA CUTTER UP" := "BA040AZSBK23.02";
	        "BK23"."X16-1.SEPA DETECT SENSOR" := "BA040AZSBK23.06";
	        "BK23"."X10-2.CLAMP&CUTTER Z-AXIS HOME SENSOR" := "Sensor".EM7[13];
	        "BK23"."X12-2.SEPA CUTTER DOWN" := "BA040AZSBK23.12";
	    END_REGION
	    REGION BK24
	        "BK24"."X10-1.SEPA CLAMP TOP REAR UP" := "BA040AZSBK24.00";
	        "BK24"."X12-1.SEPA CLAMP TOP FRONT UP" := "BA040AZSBK24.02";
	        "BK24"."X14-1.SEPA CLAMP BTM REAR UP" := "BA040AZSBK24.04";
	        "BK24"."X16-1.SEPA CLAMP BTM FRONT UP" := "BA040AZSBK24.06";
	        "BK24"."X10-2.SEPA CLAMP TOP REAR DOWN" := "BA040AZSBK24.10";
	        "BK24"."X12-2.SEPA CLAMP TOP FRONT DOWN" := "BA040AZSBK24.12";
	        "BK24"."X14-2.SEPA CLAMP BTM REAR DOWN" := "BA040AZSBK24.14";
	        "BK24"."X16-2.SEPA CLAMP BTM FRONT DOWN" := "BA040AZSBK24.16";
	    END_REGION
	    REGION BK25
	        "BK25"."X10-1.JR WINDER REAR Y-AXIS LIMIT SENSOR(-)" := "Sensor".EM7[14];
	        "BK25"."X10-2.JR WINDER REAR Y-AXIS HOME SENSOR" := "Sensor".EM7[15];
	        "BK25"."X12-1.JR WINDER REAR Y-AXIS LIMIT SENSOR(+)" := "Sensor".EM7[16];
	        "BK25"."X14-1.JR WINDER FRONT Y-AXIS LIMIT SENSOR(-)" := "Sensor".EM7[17];
	        "BK25"."X14-2.JR WINDER FRONT Y-AXIS HOME SENSOR" := "Sensor".EM7[18];
	        "BK25"."X16-1.JR WINDER FRONT Y-AXIS LIMIT SENSOR(+)" := "Sensor".EM7[20];
	    END_REGION
	    REGION BK26
	        "BK26"."X10-1.JR WINDER B-AXIS HOME SENSOR" := "Sensor".EM7[19];
	        "BK26"."X11-1.JR WINDER CLAMP TOP REAR UP/DOWN" := "BA040AZSBK26.01";
	        "BK26"."X13-1.JR WINDER CLAMP TOP FRONT UP/DOWN" := "BA040AZSBK26.03";
	        "BK26"."X15-1.JR WINDER CLAMP TOP REAR PRESSURE SWITCH" := "BA040AZSBK26.05";
	        "BK26"."X11-2.SPARE" := "BA040AZSBK26.11";
	        "BK26"."X13-2.SPARE" := "BA040AZSBK26.13";
	        "BK26"."X15-2.JR WINDER CLAMP TOP FRONT PRESSURE SWITCH" := "BA040AZSBK26.15";
	    END_REGION
	    REGION BK27
	        "BK27"."X11-1.JR WINDER CLAMP BTM REAR UP/DOWN" := "BA040AZSBK27.01";
	        "BK27"."X13-1.JR WINDER CLAMP BTM FRONT UP/DOWN" := "BA040AZSBK27.03";
	        "BK27"."X15-1.JR WINDER CLAMP FRONT TOP PRESSURE SWITCH" := "BA040AZSBK27.05";
	        "BK27"."X16-1.JR WINDER STACK DETECT SENSOR" := "BA040AZSBK27.06";
	        "BK27"."X11-2.SPARE" := "BA040AZSBK27.11";
	        "BK27"."X13-2.SPARE" := "BA040AZSBK27.13";
	        "BK27"."X15-2.JR WINDER CLAMP FRONT BTM PRESSURE SWITCH" := "BA040AZSBK27.15";
	    END_REGION
	    REGION BK28
	        "BK28"."X12-1.PUSH ROLLER BACKWARD" := "BA040AZSBK28.02";
	        "BK28"."X12-2.PUSH ROLLER FORWARD" := "BA040AZSBK28.03";
	    END_REGION
	    REGION BK29
	        "BK29"."X10-1.SUCTION PAD TOP LEFT VACUUM ON" := "BA040AZSBK29.00";
	        "BK29"."X10-2.SUCTION PAD TOP LEFT VACUUM OFF" := "BA040AZSBK29.01";
	        "BK29"."X12-1.SUCTION PAD TOP RIGHT VACUUM ON" := "BA040AZSBK29.02";
	        "BK29"."X12-2.SUCTION PAD TOP RIGHT VACUUM OFF" := "BA040AZSBK29.03";
	        "BK29"."X14-1.SUCTION PAD BTM LEFT VACUUM ON" := "BA040AZSBK29.04";
	        "BK29"."X14-2.SUCTION PAD BTM LEFT VACUUM OFF" := "BA040AZSBK29.05";
	        "BK29"."X16-1.SUCTION PAD BTM RIGHT VACUUM ON" := "BA040AZSBK29.06";
	        "BK29"."X16-2.SUCTION PAD BTM RIGHT VACUUM OFF" := "BA040AZSBK29.07";
	    END_REGION
	    REGION BK30
	        "BK30"."X10-1.SUCTION PAD TOP TAPE VACUUM ON" := "BA040AZSBK30.00";
	        "BK30"."X10-2.SUCTION PAD TOP TAPE VACUUM OFF" := "BA040AZSBK30.01";
	        "BK30"."X12-1.SUCTION PAD BTM TAPE VACUUM ON" := "BA040AZSBK30.02";
	        "BK30"."X12-2.SUCTION PAD BTM TAPE VACUUM OFF" := "BA040AZSBK30.03";
	        "BK30"."X14-1.STACK TABLE VACUUM ON" := "BA040AZSBK30.04";
	        "BK30"."X14-2.STACK TABLE VACUUM OFF" := "BA040AZSBK30.05";
	    END_REGION
	    REGION BK31
	        "BK31"."X10-1.ANODE MAIN P&P1-1 VACUUM ON" := "BA040AZSBK31.00";
	        "BK31"."X10-2.ANODE MAIN P&P1-1 VACUUM OFF" := "BA040AZSBK31.01";
	        "BK31"."X12-1.ANODE MAIN P&P2-1 VACUUM ON" := "BA040AZSBK31.02";
	        "BK31"."X12-2.ANODE MAIN P&P2-1 VACUUM OFF" := "BA040AZSBK31.03";
	        "BK31"."X14-1.ANODE MAIN NG P&P VACUUM ON" := "BA040AZSBK31.04";
	        "BK31"."X14-2.ANODE MAIN NG P&P VACUUM OFF" := "BA040AZSBK31.05";
	        "BK31"."X16-1.ANODE ALIGN TABLE VACUUM ON" := "BA040AZSBK31.06";
	        "BK31"."X16-2.ANODE ALIGN TABLE VACUUM OFF" := "BA040AZSBK31.07";
	    END_REGION
	    REGION BK32
	        "BK32"."X10-1.CATHODE MAIN P&P1-1 VACUUM ON" := "BA040AZSBK32.00";
	        "BK32"."X10-2.CATHODE MAIN P&P1-1 VACUUM OFF" := "BA040AZSBK32.01";
	        "BK32"."X12-1.CATHODE MAIN P&P2-1 VACUUM ON" := "BA040AZSBK32.02";
	        "BK32"."X12-2.CATHODE MAIN P&P2-1 VACUUM OFF" := "BA040AZSBK32.03";
	        "BK32"."X14-1.CATHODE MAIN NG P&P VACUUM ON" := "BA040AZSBK32.04";
	        "BK32"."X14-2.CATHODE MAIN NG P&P VACUUM OFF" := "BA040AZSBK32.05";
	        "BK32"."X16-1.CATHODE ALIGN TABLE VACUUM ON" := "BA040AZSBK32.06";
	        "BK32"."X16-2.CATHODE ALIGN TABLE VACUUM OFF" := "BA040AZSBK32.07";
	    END_REGION
	    REGION BK33
	        "BK33"."X10-1.ANODE MAIN P&P1-2 VACUUM ON" := "BA040AZSBK33.00";
	        "BK33"."X10-2.ANODE MAIN P&P1-2 VACUUM OFF" := "BA040AZSBK33.01";
	        "BK33"."X12-1.CATHODE MAIN P&P1-2 VACUUM ON" := "BA040AZSBK33.02";
	        "BK33"."X12-2.CATHODE MAIN P&P1-2 VACUUM OFF" := "BA040AZSBK33.03";
	        "BK33"."X14-1.ANODE MAIN P&P2-2 VACUUM ON" := "BA040AZSBK33.04";
	        "BK33"."X14-2.ANODE MAIN P&P2-2 VACUUM OFF" := "BA040AZSBK33.05";
	        "BK33"."X16-1.CATHODE MAIN P&P2-2 VACUUM ON" := "BA040AZSBK33.06";
	        "BK33"."X16-2.CATHODE MAIN P&P2-2 VACUUM OFF" := "BA040AZSBK33.07";
	    END_REGION
	    
	    REGION SBK
	    REGION SBK01
	        "SBK01"."EMO01 CH.A" := "BA040AZSSBK01.00";
	        "SBK01"."EMO02 CH.A" := "BA040AZSSBK01.01";
	        "SBK01"."EMO04 CH.A" := "BA040AZSSBK01.03";
	    END_REGION
	    REGION SBK02
	        "SBK02"."SCS BOX SCS MODE SLELECT SS.SETUP" := "BA040AZSSBK02.00";
	        "SBK02"."SCS BOX SCS MODE SLELECT SS.DISABLE" := "BA040AZSSBK02.01";
	        "SBK02"."EMO05 CH.A" := "BA040AZSSBK02.02";
	        "SBK02"."SCS BOX SCS MODE SLELECT SS.AUTO" := "BA040AZSSBK02.04";
	        "SBK02"."SCS BOX SCS MODE SELECT PL.PENDANT" := "BA040AZSSBK02.10";
	        "SBK02"."SCS BOX SCS MODE SELECT PL.DISABLE" := "BA040AZSSBK02.11";
	    END_REGION
	    REGION SBK03
	        "SBK03"."ROLL CHANGE TOP SS.AUTO" := "BA040AZSSBK03.00";
	        "SBK03"."ROLL CHANGE BTM SS.AUTO" := "BA040AZSSBK03.01";
	        "SBK03"."ROLL CHANGE TOP SS.CHANGE" := "BA040AZSSBK03.04";
	        "SBK03"."ROLL CHANGE BTM SS.CHANGE" := "BA040AZSSBK03.05";
	        "SBK03"."ROLL CHANGE LH IN PROGRESS" := "BA040AZSSBK03.10";
	        "SBK03"."ROLL CHANGE RH IN PROGRESS" := "BA040AZSSBK03.11";
	    END_REGION
	    REGION SBK04
	        "SBK04"."GATE EC U/W MAIN PB.LOCK" := "BA040AZSSBK04.00";
	        "SBK04"."GATE EC U/W MAIN PB.RESET" := "BA040AZSSBK04.01";
	        "SBK04"."GATE EC U/W MAIN PB.UNLOCK" := "BA040AZSSBK04.04";
	        "SBK04"."GATE EC U/W MAIN PL.LOCK" := "BA040AZSSBK04.10";
	        "SBK04"."GATE EC U/W MAIN PL.UNLOCK" := "BA040AZSSBK04.11";
	        "SBK04"."GATE EC U/W MAIN PL.RESET" := "BA040AZSSBK04.12";
	    END_REGION
	    REGION SBK05
	        "SBK05"."GATE EC U/W TOP PB.LOCK" := "BA040AZSSBK05.00";
	        "SBK05"."GATE EC U/W TOP PB.RESET" := "BA040AZSSBK05.01";
	        "SBK05"."GATE EC U/W TOP PB.UNLOCK" := "BA040AZSSBK05.04";
	        "SBK05"."GATE EC U/W TOP PL.LOCK" := "BA040AZSSBK05.10";
	        "SBK05"."GATE EC U/W TOP PL.UNLOCK" := "BA040AZSSBK05.11";
	        "SBK05"."GATE EC U/W TOP PL.RESET" := "BA040AZSSBK05.12";
	    END_REGION
	    REGION SBK06
	        "SBK06"."GATE EC U/W BTM PB.LOCK" := "BA040AZSSBK06.00";
	        "SBK06"."GATE EC U/W BTM PB.RESET" := "BA040AZSSBK06.01";
	        "SBK06"."GATE EC U/W BTM PB.UNLOCK" := "BA040AZSSBK06.04";
	        "SBK06"."GATE EC U/W BTM PL.LOCK" := "BA040AZSSBK06.10";
	        "SBK06"."GATE EC U/W BTM PL.UNLOCK" := "BA040AZSSBK06.11";
	        "SBK06"."GATE EC U/W BTM PL.RESET" := "BA040AZSSBK06.12";
	    END_REGION
	    REGION SBK07
	        "SBK07"."GATE EC SCRAP BOX-1 PB.LOCK" := "BA040AZSSBK07.00";
	        "SBK07"."GATE EC SCRAP BOX-1 PB.RESET" := "BA040AZSSBK07.01";
	        "SBK07"."GATE EC SCRAP BOX-1 PB.UNLOCK" := "BA040AZSSBK07.04";
	        "SBK07"."GATE EC SCRAP BOX-1 PL.LOCK" := "BA040AZSSBK07.10";
	        "SBK07"."GATE EC SCRAP BOX-1 PL.UNLOCK" := "BA040AZSSBK07.11";
	        "SBK07"."GATE EC SCRAP BOX-1 PL.RESET" := "BA040AZSSBK07.12";
	    END_REGION
	    REGION SBK08
	        "SBK08"."SAFETY DOOR LOCK1.INPUT" := "BA040AZSSBK08.00";
	        "SBK08"."SAFETY DOOR LOCK2.INPUT" := "BA040AZSSBK08.01";
	        "SBK08"."SAFETY DOOR LOCK3.INPUT" := "BA040AZSSBK08.02";
	        "SBK08"."SAFETY DOOR LOCK1.OUTPUT" := "BA040AZSSBK08.10";
	        "SBK08"."SAFETY DOOR LOCK2.OUTPUT" := "BA040AZSSBK08.11";
	        "SBK08"."SAFETY DOOR LOCK3.OUTPUT" := "BA040AZSSBK08.12";
	    END_REGION
	    REGION SBK09
	        "SBK09"."SAFETY DOOR LOCK4.INPUT" := "BA040AZSSBK09.00";
	        "SBK09"."SAFETY DOOR LOCK5.INPUT" := "BA040AZSSBK09.01";
	        "SBK09"."SAFETY DOOR LOCK6.INPUT" := "BA040AZSSBK09.02";
	        "SBK09"."SAFETY DOOR LOCK4.OUTPUT" := "BA040AZSSBK09.10";
	        "SBK09"."SAFETY DOOR LOCK5.OUTPUT" := "BA040AZSSBK09.11";
	        "SBK09"."SAFETY DOOR LOCK6.OUTPUT" := "BA040AZSSBK09.12";
	    END_REGION
	    REGION SBK10
	        "SBK10"."SAFETY DOOR LOCK7.INPUT" := "BA040AZSSBK10.00";
	        "SBK10"."SAFETY DOOR LOCK8.INPUT" := "BA040AZSSBK10.01";
	        "SBK10"."SAFETY DOOR LOCK7.OUTPUT" := "BA040AZSSBK10.10";
	        "SBK10"."SAFETY DOOR LOCK8.OUTPUT" := "BA040AZSSBK10.11";
	    END_REGION
	    REGION SBK11
	        "SBK11"."GATE EC SCRAP BOX-2 PB.LOCK" := "BA040AZSSBK11.00";
	        "SBK11"."GATE EC SCRAP BOX-2 PB.RESET" := "BA040AZSSBK11.01";
	        "SBK11"."GATE EC SCRAP BOX-2 PB.UNLOCK" := "BA040AZSSBK11.04";
	        "SBK11"."GATE EC SCRAP BOX-2 PL.LOCK" := "BA040AZSSBK11.10";
	        "SBK11"."GATE EC SCRAP BOX-2 PL.UNLOCK" := "BA040AZSSBK11.11";
	        "SBK11"."GATE EC SCRAP BOX-2 PL.RESET" := "BA040AZSSBK11.12";
	    END_REGION
	    REGION SBK12
	        "SBK12"."ANODE CONVEYOR COVER BACKWARD" := "BA040AZSSBK12.00";
	        "SBK12"."CATHODE CONVEYOR COVER BACKWARD" := "BA040AZSSBK12.01";
	        "SBK12"."ANODE CONVEYOR COVER FORWARD" := "BA040AZSSBK12.04";
	        "SBK12"."CATHODE CONVEYOR COVER FORWARD" := "BA040AZSSBK12.05";
	    END_REGION
	    REGION SBK13
	        "SBK13"."SAFETY DOOR LOCK10.INPUT" := "BA040AZSSBK13.00";
	        "SBK13"."SAFETY DOOR LOCK12.INPUT" := "BA040AZSSBK13.02";
	        "SBK13"."SAFETY DOOR LOCK10.OUTPUT" := "BA040AZSSBK13.10";
	        "SBK13"."SAFETY DOOR LOCK12.OUTPUT" := "BA040AZSSBK13.12";
	    END_REGION
	    END_REGION
	    REGION PM
	        "PM01"."SEPA DANCER FORWARD" := "BA040AZSPM01.00";
	        "PM01"."SEPA DANCER BACKWARD" := "BA040AZSPM01.01";
	        "PM01"."SEPA UW #1 IONIZER TOP ON" := "BA040AZSPM01.02";
	        "PM01"."SEPA UW #1 IONIZER BTM ON" := "BA040AZSPM01.04";
	        "PM01"."SEPA UW #1 AIR SHAFT TOP ON" := "BA040AZSPM01.06";
	        "PM01"."SEPA UW #1 AIR SHAFT TOP OFF" := "BA040AZSPM01.07";
	        "PM01"."SEPA UW #1 AIR SHAFT BTM ON" := "BA040AZSPM01.10";
	        "PM01"."SEPA UW #1 AIR SHAFT BTM OFF" := "BA040AZSPM01.11";
	        //"PM01".SPARE_3 := "BA030AZSPM01.10";
	        //"PM01".SPARE_4 := "BA030AZSPM01.11";
	        "PM01"."ANODE CONVEYOR PICK UP BLOWER ON/OFF" := "BA040AZSPM01.14";
	        "PM01"."CATHODE CONVEYOR PICK UP BLOWER ON/OFF" := "BA040AZSPM01.16";
	    END_REGION
	    REGION PM02
	        "PM02"."SUCTION PAD #1 TOP UP" := "BA040AZSPM02.00";
	        "PM02"."SUCTION PAD #1 TOP DOWN" := "BA040AZSPM02.01";
	        "PM02"."SUCTION PAD #1 BTM UP" := "BA040AZSPM02.02";
	        "PM02"."SUCTION PAD #1 BTM DOWN" := "BA040AZSPM02.03";
	        "PM02"."CUTTER #1 UP" := "BA040AZSPM02.04";
	        "PM02"."CUTTER #1 DOWN" := "BA040AZSPM02.05";
	        "PM02"."TAPE #1 TOP UP" := "BA040AZSPM02.06";
	        "PM02"."TAPE #1 TOP DOWN" := "BA040AZSPM02.07";
	        "PM02"."TAPE #1 BTM UP" := "BA040AZSPM02.10";
	        "PM02"."TAPE #1 BTM DOWN" := "BA040AZSPM02.11";
	        "PM02"."SPLICE HEAD ROTATE #1 TOP FORWARD" := "BA040AZSPM02.12";
	        "PM02"."SPLICE HEAD ROTATE #1 TOP BACKWARD" := "BA040AZSPM02.13";
	        "PM02"."SPLICE HEAD ROTATE #1 BTM FORWARD" := "BA040AZSPM02.14";
	        "PM02"."SPLICE HEAD ROTATE #1 BTM BACKWARD" := "BA040AZSPM02.15";
	    END_REGION
	    REGION PM03
	        "PM03"."SEPA CUTTER REAR UP / SEPA CUTTER FRONT UP" := "BA040AZSPM03.00";
	        "PM03"."SEPA CUTTER REAR DOWN / SEPA CUTTER FRONT DOWN" := "BA040AZSPM03.01";
	        "PM03"."SEPA CLAMP TOP REAR UP" := "BA040AZSPM03.02";
	        "PM03"."SEPA CLAMP TOP REAR DOWN" := "BA040AZSPM03.03";
	        "PM03"."SEPA CLAMP TOP FRONT UP" := "BA040AZSPM03.04";
	        "PM03"."SEPA CLAMP TOP FRONT DOWN" := "BA040AZSPM03.05";
	        "PM03"."SEPA CLAMP BTM REAR UP" := "BA040AZSPM03.06";
	        "PM03"."SEPA CLAMP BTM REAR DOWN" := "BA040AZSPM03.07";
	        "PM03"."SEPA CLAMP BTM FRONT UP" := "BA040AZSPM03.10";
	        "PM03"."SEPA CLAMP BTM FRONT DOWN" := "BA040AZSPM03.11";
	        "PM03"."SEPA GRIPPER OPEN" := "BA040AZSPM03.12";
	        "PM03"."SEPA GRIPPER  CLOSE" := "BA040AZSPM03.13";
	        "PM03"."SEPA GRIPPER FORWARD" := "BA040AZSPM03.14";
	        "PM03"."SEPA GRIPPER BACKWARD" := "BA040AZSPM03.15";
	    END_REGION
	    REGION PM04
	        "PM04"."STACK TABLE GAP PAD UP" := "BA040AZSPM04.00";
	        "PM04"."STACK TABLE GAP PAD DOWN" := "BA040AZSPM04.01";
	        "PM04"."CATHODE MANDREL CLAMP FRONT ON" := "BA040AZSPM04.02";
	        "PM04"."CATHODE MANDREL CLAMP REAR ON" := "BA040AZSPM04.04";
	        "PM04"."ANODE MANDREL CLAMP FRONT ON" := "BA040AZSPM04.06";
	        "PM04"."ANODE MANDREL CLAMP REAR ON" := "BA040AZSPM04.10";
	    END_REGION
	    REGION PM05
	        "PM05"."ANODE GLASS CLEANING ON" := "BA040AZSPM05.00";
	        "PM05"."ANODE MAIN NG P&P UP" := "BA040AZSPM05.02";
	        "PM05"."ANODE MAIN NG P&P DOWN" := "BA040AZSPM05.03";
	        "PM05"."ANODE MAIN NG P&P 1st FORWARD" := "BA040AZSPM05.04";
	        "PM05"."ANODE MAIN NG P&P 1st BACKWARD" := "BA040AZSPM05.05";
	        "PM05"."ANODE MAIN NG P&P 2nd FORWARD" := "BA040AZSPM05.06";
	        "PM05"."ANODE MAIN NG P&P 2nd BACKWARD" := "BA040AZSPM05.07";
	        "PM05"."ANODE FIX FRONT FORWARD / ANODE FIX REAR FORWARD" := "BA040AZSPM05.10";
	        "PM05"."ANODE FIX FRONT BACKWARD / ANODE FIX REAR BACKWARD" := "BA040AZSPM05.11";
	        "PM05"."ANODE MAIN P&P#1 Rotary CW" := "BA040AZSPM05.12";
	        "PM05"."ANODE MAIN P&P#1 Rotary CCW" := "BA040AZSPM05.13";
	        "PM05"."ANODE NG BOX LIFT UP" := "BA040AZSPM05.14";
	        "PM05"."ANODE NG BOX LIFT DOWN" := "BA040AZSPM05.15";
	        "PM05"."ANODE NG BOX LOCK UP" := "BA040AZSPM05.16";
	        "PM05"."ANODE NG BOX LOCK DOWN" := "BA040AZSPM05.17";
	    END_REGION
	    REGION PM06
	        "PM06"."CATHODE GLASS CLEANING ON" := "BA040AZSPM06.00";
	        "PM06"."CATHODE MAIN NG P&P UP" := "BA040AZSPM06.02";
	        "PM06"."CATHODE MAIN NG P&P DOWN" := "BA040AZSPM06.03";
	        "PM06"."CATHODE MAIN NG P&P 1st FORWARD" := "BA040AZSPM06.04";
	        "PM06"."CATHODE MAIN NG P&P 1st BACKWARD" := "BA040AZSPM06.05";
	        "PM06"."CATHODE MAIN NG P&P 2nd FORWARD" := "BA040AZSPM06.06";
	        "PM06"."CATHODE MAIN NG P&P 2nd BACKWARD" := "BA040AZSPM06.07";
	        "PM06"."CATHODE FIX FRONT FORWARD / CATHODE FIX REAR FORWARD" := "BA040AZSPM06.10";
	        "PM06"."CATHODE FIX FRONT BACKWARD / CATHODE FIX REAR BACKWARD" := "BA040AZSPM06.11";
	        "PM06"."CATHODE MAIN P&P#1 Rotary CW" := "BA040AZSPM06.12";
	        "PM06"."CATHODE MAIN P&P#1 Rotary CCW" := "BA040AZSPM06.13";
	        "PM06"."CATHODE NG BOX LIFT UP" := "BA040AZSPM06.14";
	        "PM06"."CATHODE NG BOX LIFT DOWN" := "BA040AZSPM06.15";
	        "PM06"."CATHODE NG BOX LOCK UP" := "BA040AZSPM06.16";
	        "PM06"."CATHODE NG BOX LOCK DOWN" := "BA040AZSPM06.17";
	    END_REGION
	    REGION PM07
	        "PM07"."JR WINDER CLAMP TOP REAR  UP" := "BA040AZSPM07.00";
	        "PM07"."JR WINDER CLAMP TOP REAR  DOWN" := "BA040AZSPM07.01";
	        "PM07"."JR WINDER CLAMP BTM REAR UP" := "BA040AZSPM07.02";
	        "PM07"."JR WINDER CLAMP BTM REAR DOWN" := "BA040AZSPM07.03";
	        "PM07"."JR WINDER CLAMP TOP FRONT UP" := "BA040AZSPM07.04";
	        "PM07"."JR WINDER CLAMP TOP FRONT DOWN" := "BA040AZSPM07.05";
	        "PM07"."JR WINDER CLAMP BTM FRONT UP" := "BA040AZSPM07.06";
	        "PM07"."JR WINDER CLAMP BTM FRONT DOWN" := "BA040AZSPM07.07";
	        //"PM07".SPARE := "BA030AZSPM07.08";
	        //"PM07".SPARE_1 := "BA030AZSPM07.09";
	        "PM07"."PUSH ROLLER FORWARD" := "BA040AZSPM07.12";
	        "PM07"."PUSH ROLLER BACKWARD" := "BA040AZSPM07.13";
	        "PM07"."ANODE CONVEYOR COVER FORWARD" := "BA040AZSPM07.14";
	        "PM07"."ANODE CONVEYOR COVER BACKWARD" := "BA040AZSPM07.15";
	        "PM07"."CATHODE CONVEYOR COVER FORWARD" := "BA040AZSPM07.16";
	        "PM07"."CATHODE CONVEYOR COVER BACKWARD" := "BA040AZSPM07.17";
	    END_REGION
	END_REGION
	REGION SP500
	    REGION SP501
	        "SP501"."CONTROL DC POWER TRIPPED E156CB" := "BA040AZSSP501.00";
	        "SP501"."SAFETY DC POWER TRIPPED E218CB" := "BA040AZSSP501.01";
	        "SP501"."CLASS 2 SMPS POWER TRIPPED E308CB" := "BA040AZSSP501.02";
	        "SP501"."CLASS 2 SMPS MONITORING E310PWS" := "BA040AZSSP501.03";
	        "SP501"."ET200ECO PN-1 POWER TRIPPED E324CB" := "BA040AZSSP501.04";
	        "SP501"."ET200ECO PN-2 POWER TRIPPED E328CB" := "BA040AZSSP501.05";
	        "SP501"."ET200ECO PN-3 POWER TRIPPED E332CB" := "BA040AZSSP501.06";
	        "SP501"."ET200ECO PN-4 POWER TRIPPED E336CB" := "BA040AZSSP501.07";
	        "SP501"."SEPA UW IONIZER TOP MAINTERNANCE DETECTION" := "BA040AZSSP501.10";
	        "SP501"."SEPA UW IONIZER TOP ERROR" := "BA040AZSSP501.11";
	        "SP501"."SEPA UW IONIZER BOTTOM MAINTERNANCE DETECTION" := "BA040AZSSP501.14";
	        "SP501"."SEPA UW IONIZER BOTTOM ERROR" := "BA040AZSSP501.15";
	    END_REGION
	    REGION SP502
	        "SP502"."CLASS2 SMPS ALARM RESET" := "BA040AZSSP502.00";
	        "SP502"."SEPA UW IONIZER TOP MAINTERNANCE DETECTION" := "BA040AZSSP502.10";
	        "SP502"."SEPA UW IONIZER TOP DISCHARGE STOP" := "BA040AZSSP502.11";
	        "SP502"."SEPA UW IONIZER BOTTOM MAINTERNANCE DETECTION" := "BA040AZSSP502.14";
	        "SP502"."SEPA UW IONIZER BOTTOM DISCHARGE STOP" := "BA040AZSSP502.15";
	    END_REGION
	    REGION SP506
	        "SP506"."PHMI EMERGENCY STOP CH.A" := "BA040AZSSP506.00";
	        "SP506"."PHMI ENABLE SWITCH CH.A" := "BA040AZSSP506.01";
	        "SP506"."PHMI EMERGENCY STOP CH.B" := "BA040AZSSP506.04";
	        "SP506"."PHMI ENABLE SWITCH CH.B" := "BA040AZSSP506.05";
	    END_REGION
	    REGION SP507
	        "SP507"."UNWINDER EPCC01 INTERLOCK" := "BA040AZSSP507.00";
	        "SP507"."UNWINDER EPCC02 INTERLOCK" := "BA040AZSSP507.01";
	        "SP507"."UNWINDER EPCC03 INTERLOCK" := "BA040AZSSP507.02";
	        "SP507"."UNWINDER EPCC04 INTERLOCK" := "BA040AZSSP507.03";
	    END_REGION
	    REGION SP508
	        "SP508"."ANODE ALIGN VISION BUSY (STO)" := "BA030AZSSP508.00";
	        "SP508"."ANODE ALIGN VISION RESULT (OK)" := "BA030AZSSP508.01";
	        "SP508"."STACK VISION BUSY (STO)" := "BA030AZSSP508.02";
	        "SP508"."STACK VISION RESULT (OK)" := "BA030AZSSP508.03";
	        "SP508"."CATHODE ALIGN VISION BUSY (STO)" := "BA030AZSSP508.04";
	        "SP508"."CATHODE ALIGN VISION RESULT (OK)" := "BA030AZSSP508.05";
	    END_REGION
	END_REGION
	REGION SP200
	    REGION SP201
	        "SP201"."MAIN OP AUTO INITIATE PBL (GREEN)" := "BA040AZSSP201.00";
	        "SP201"."MAIN OP STOP PBL (RED)" := "BA040AZSSP201.01";
	        "SP201"."MAIN HMI POWER TRIPPED E110CB" := "BA040AZSSP201.10";
	    END_REGION
	    REGION SP202
	        "SP202"."AUTO INITIATE PBL LAMP (GREEN)" := "BA040AZSSP202.00";
	        "SP202"."STOP PBL LAMP ON (RED)" := "BA040AZSSP202.01";
	        "SP202"."ENABLE PBL LAMP ON (BLACK)" := "BA040AZSSP202.03";
	        "SP202"."SAFETY RESET PBL LAMP (BLUE)" := "BA040AZSSP202.04";
	        "SP202"."TOWER LAMP 1 ON (RED)" := "BA040AZSSP202.10";
	        "SP202"."TOWER LAMP 2 ON (AMBER)" := "BA040AZSSP202.11";
	        "SP202"."TOWER LAMP 3 ON (GREEN)" := "BA040AZSSP202.12";
	        "SP202"."TOWER LAMP 4 ON (WHITE)" := "BA040AZSSP202.13";
	        "SP202"."TOWER LAMP 5 ON (BLUE)" := "BA040AZSSP202.14";
	        "SP202"."Buzzer On" := "BA040AZSSP202.15";
	        //"SP202"."TOWER LAMP BUZZER ON" := "BA030AZSSP202.15";
	    END_REGION
	    REGION SP203
	        "SP203"."MODE SELECT AUTO" := "BA040AZSSP203.00";
	        "SP203"."HOME PBL (GREEN)" := "BA040AZSSP203.01";
	        "SP203"."SAFETY RESET PBL (BLUE)" := "BA040AZSSP203.02";
	        "SP203"."SCS MODE SELECT AUTO" := "BA040AZSSP203.03";
	        "SP203"."MODE SELECT MANUAL" := "BA040AZSSP203.04";
	        "SP203"."ENABLE PBL (BLACK)" := "BA040AZSSP203.05";
	        "SP203"."SCS MODE SELECT SETUP" := "BA040AZSSP203.06";
	        "SP203"."SCS MODE SELECT DISABLE" := "BA040AZSSP203.07";
	    END_REGION
	    REGION SP204
	        "SP204"."MAIN OP EMERGENCY STOP CH.A" := "BA040AZSSP204.00";
	        "SP204"."MAIN OP EMERGENCY STOP CH.B" := "BA040AZSSP204.04";
	    END_REGION
	    REGION SP205
	        "SP205"."PENDANT REQUIRED PL (YELLOW)" := "BA040AZSSP205.00";
	        "SP205"."HOME PBL LAMP ON (GREEN)" := "BA040AZSSP205.02";
	        "SP205"."SCS SELECT DISABLE PL (GREEN)" := "BA040AZSSP205.07";
	    END_REGION
	END_REGION
	
	
	
	
	
	
	
	
	
	
	
	
	
	
	
	
	
	
	
	
	
	
	
	
	
	
	
	
	
	
	
	
	
	
	
	
	
	
	
	
	
	
	
	
	
	
	
	
	
	
	
	
	
	
	
	
	
	
	
	
	
	
	
	
	
	
	
	
	
	
	
	
	
	
	
	
	
	
	
END_FUNCTION

FUNCTION_BLOCK "CallInterfaceSignals"   // FB38, LAD
TITLE = CallInterfaceSignals
AUTHOR : SICAR
FAMILY : Diag
VERSION : 1.0
// Der Baustein dient als Aufrufschnittstelle für den Funktionsbaustein „LSicar_InterfaceSignalsBool“. Er ist als Funktionsbaustein ausgeführt, um die intern aufgerufenen FBs mittels Multiinstanzen realisieren zu können.  
// Die Funktionsbausteine und das zugehörige WinCC-Bild sind für 16 Signaldatensätze („Schnittstelle Signale 01“ … „Schnittstellen Signale 16“) mit jeweils 32 boolschen Signalen vorgesehen.  
// 
// **PLC-Datentypen**  
//  LSicar_typeInterfaceSignalsBool 
//  typeInterfaceSignalsHmi 
//  LSicar _typeInterfaceSignals 
// 
// **WinCC-Diagnosebild**  
// 
// ![Icon](_Icon/reference.PNG)
// 
// siehe ..\Library Types\LSicar_InterfaceSignalsBool.pdf  
// 
//  
// 
// **Beispielaufruf**  
// Abbildung in Kontaktplan (KOP).  D:\Software\Symbols_Icons\BMPs-JPGs-PNGs\Verschiedene\symb_user_goto_transparent.pngEin lauffähiger Programm-Aufruf hierzu ist im „SICAR-StartUp“-Projekt enthalten.  
// 
// **Aufrufschnittstelle**  
// Der Baustein wird einmalig im zyklischen Programm aufgerufen.  
// 
// **Intern verwendete „Erweiterte Anweisungen / Bausteine“**  
// ..\Library Types\LSicar_InterfaceSignalsBool.pdf
// The block serves as a calling interface of the block “InterfaceSignalsBool“. The block is designed as function block in order to implement the block calls as multi-instances.
// stored: IsIECCheckEnabled true, MemoryReserve 100, SetENOAutomatically true
   VAR
      statReadValueHmi : Bool;   // HMI: Lese Signalwert / HMI: Read value signal
      statSelectSignalsHmi : USInt := 1;   // HMI: Angewählte Interface Schnittstelle (1..16) / HMI: Selected interface signals (1..16)
      statSelectSignalsOld { ExternalAccessible := 'False'; ExternalVisible := 'False'; ExternalWritable := 'False'} : USInt;   // Altwert: Angewählte Interface Schnittstelle / Old value: Selected interface signals
      statRisEdgeReadName { ExternalAccessible := 'False'; ExternalVisible := 'False'; ExternalWritable := 'False'} : Bool;   // Steigende Flanke / Rising edge
      statPosPulseReadName : Bool;   // Positiver Impuls / Positive pulse
      statInterfaceSignalsHmi : Array[0..99] of "typeInterfaceSignalsHmi";   // HMI: Beschreibung, Wert und Symbolischer Name / HMI: Description, value and symbolic name
      instSignals1Left { S7_SetPoint := 'True'} : "LAF_InterfaceSignalsBool";
      instSignals1Right { S7_SetPoint := 'True'} : "LAF_InterfaceSignalsBool";
      instSignals2Left { S7_SetPoint := 'True'} : "LAF_InterfaceSignalsBool";
      instSignals2Right { S7_SetPoint := 'True'} : "LAF_InterfaceSignalsBool";
      instSignals3Left { S7_SetPoint := 'True'} : "LAF_InterfaceSignalsBool";
      instSignals3Right { S7_SetPoint := 'True'} : "LAF_InterfaceSignalsBool";
      instSignals4Left { S7_SetPoint := 'True'} : "LAF_InterfaceSignalsBool";
      instSignals4Right { S7_SetPoint := 'True'} : "LAF_InterfaceSignalsBool";
      instSignals5Left { S7_SetPoint := 'True'} : "LAF_InterfaceSignalsBool";
      instSignals5Right { S7_SetPoint := 'True'} : "LAF_InterfaceSignalsBool";
      instSignals6Left { S7_SetPoint := 'True'} : "LAF_InterfaceSignalsBool";
      instSignals6Right { S7_SetPoint := 'True'} : "LAF_InterfaceSignalsBool";
      instSignals7Left { S7_SetPoint := 'True'} : "LAF_InterfaceSignalsBool";
      instSignals7Right { S7_SetPoint := 'True'} : "LAF_InterfaceSignalsBool";
      instSignals8Left { S7_SetPoint := 'True'} : "LAF_InterfaceSignalsBool";
      instSignals8Right { S7_SetPoint := 'True'} : "LAF_InterfaceSignalsBool";
      instSignals9Left { S7_SetPoint := 'True'} : "LAF_InterfaceSignalsBool";
      instSignals9Right { S7_SetPoint := 'True'} : "LAF_InterfaceSignalsBool";
      instSignals10Left { S7_SetPoint := 'True'} : "LAF_InterfaceSignalsBool";
      instSignals10Right { S7_SetPoint := 'True'} : "LAF_InterfaceSignalsBool";
      instSignals11Left { S7_SetPoint := 'True'} : "LAF_InterfaceSignalsBool";
      instSignals11Right { S7_SetPoint := 'True'} : "LAF_InterfaceSignalsBool";
      instSignals12Left { S7_SetPoint := 'True'} : "LAF_InterfaceSignalsBool";
      instSignals12Right { S7_SetPoint := 'True'} : "LAF_InterfaceSignalsBool";
      instSignals13Left { S7_SetPoint := 'True'} : "LAF_InterfaceSignalsBool";
      instSignals13Right { S7_SetPoint := 'True'} : "LAF_InterfaceSignalsBool";
      instSignals14Left { S7_SetPoint := 'True'} : "LAF_InterfaceSignalsBool";
      instSignals14Right { S7_SetPoint := 'True'} : "LAF_InterfaceSignalsBool";
      instSignals15Left { S7_SetPoint := 'True'} : "LAF_InterfaceSignalsBool";
      instSignals15Right { S7_SetPoint := 'True'} : "LAF_InterfaceSignalsBool";
      instSignals16Left { S7_SetPoint := 'True'} : "LAF_InterfaceSignalsBool";
      instSignals16Right { S7_SetPoint := 'True'} : "LAF_InterfaceSignalsBool";
      instSignals17Left { S7_SetPoint := 'True'} : "LAF_InterfaceSignalsBool";
      instSignals17Right { S7_SetPoint := 'True'} : "LAF_InterfaceSignalsBool";
      instSignals18Left { S7_SetPoint := 'True'} : "LAF_InterfaceSignalsBool";
      instSignals18Right { S7_SetPoint := 'True'} : "LAF_InterfaceSignalsBool";
      instSignals19Left { S7_SetPoint := 'True'} : "LAF_InterfaceSignalsBool";
      instSignals19Right { S7_SetPoint := 'True'} : "LAF_InterfaceSignalsBool";
      instSignals20Left { S7_SetPoint := 'True'} : "LAF_InterfaceSignalsBool";
      instSignals20Right { S7_SetPoint := 'True'} : "LAF_InterfaceSignalsBool";
      instSignals21Left { S7_SetPoint := 'True'} : "LAF_InterfaceSignalsBool";
      instSignals21Right { S7_SetPoint := 'True'} : "LAF_InterfaceSignalsBool";
      instSignals22Left { S7_SetPoint := 'True'} : "LAF_InterfaceSignalsBool";
      instSignals22Right { S7_SetPoint := 'True'} : "LAF_InterfaceSignalsBool";
      instSignals23Left { S7_SetPoint := 'True'} : "LAF_InterfaceSignalsBool";
      instSignals23Right { S7_SetPoint := 'True'} : "LAF_InterfaceSignalsBool";
      instSignals24Left { S7_SetPoint := 'True'} : "LAF_InterfaceSignalsBool";
      instSignals24Right { S7_SetPoint := 'True'} : "LAF_InterfaceSignalsBool";
      instSignals25Left { S7_SetPoint := 'True'} : "LAF_InterfaceSignalsBool";
      instSignals25Right { S7_SetPoint := 'True'} : "LAF_InterfaceSignalsBool";
      instSignals26Left { S7_SetPoint := 'True'} : "LAF_InterfaceSignalsBool";
      instSignals26Right { S7_SetPoint := 'True'} : "LAF_InterfaceSignalsBool";
      instSignals27Left { S7_SetPoint := 'True'} : "LAF_InterfaceSignalsBool";
      instSignals27Right { S7_SetPoint := 'True'} : "LAF_InterfaceSignalsBool";
      instSignals28Left { S7_SetPoint := 'True'} : "LAF_InterfaceSignalsBool";
      instSignals28Right { S7_SetPoint := 'True'} : "LAF_InterfaceSignalsBool";
      instSignals29Left { S7_SetPoint := 'True'} : "LAF_InterfaceSignalsBool";
      instSignals29Right { S7_SetPoint := 'True'} : "LAF_InterfaceSignalsBool";
      instSignals30Left { S7_SetPoint := 'True'} : "LAF_InterfaceSignalsBool";
      instSignals30Right { S7_SetPoint := 'True'} : "LAF_InterfaceSignalsBool";
      instSignals31Left { S7_SetPoint := 'True'} : "LAF_InterfaceSignalsBool";
      instSignals31Right { S7_SetPoint := 'True'} : "LAF_InterfaceSignalsBool";
      instSignals32Left { S7_SetPoint := 'True'} : "LAF_InterfaceSignalsBool";
      instSignals32Right { S7_SetPoint := 'True'} : "LAF_InterfaceSignalsBool";
      instSignals33Left { S7_SetPoint := 'True'} : "LAF_InterfaceSignalsBool";
      instSignals33Right { S7_SetPoint := 'True'} : "LAF_InterfaceSignalsBool";
      instSignals34Left { S7_SetPoint := 'True'} : "LAF_InterfaceSignalsBool";
      instSignals34Right { S7_SetPoint := 'True'} : "LAF_InterfaceSignalsBool";
      instSignals35Left { S7_SetPoint := 'True'} : "LAF_InterfaceSignalsBool";
      instSignals35Right { S7_SetPoint := 'True'} : "LAF_InterfaceSignalsBool";
      instSignals36Left { S7_SetPoint := 'True'} : "LAF_InterfaceSignalsBool";
      instSignals36Right { S7_SetPoint := 'True'} : "LAF_InterfaceSignalsBool";
      instSignals37Left { S7_SetPoint := 'True'} : "LAF_InterfaceSignalsBool";
      instSignals37Right { S7_SetPoint := 'True'} : "LAF_InterfaceSignalsBool";
      instSignals38Left { S7_SetPoint := 'True'} : "LAF_InterfaceSignalsBool";
      instSignals38Right { S7_SetPoint := 'True'} : "LAF_InterfaceSignalsBool";
      instSignals39Left { S7_SetPoint := 'True'} : "LAF_InterfaceSignalsBool";
      instSignals39Right { S7_SetPoint := 'True'} : "LAF_InterfaceSignalsBool";
      instSignals40Left { S7_SetPoint := 'True'} : "LAF_InterfaceSignalsBool";
      instSignals40Right { S7_SetPoint := 'True'} : "LAF_InterfaceSignalsBool";
      instSignals41Left { S7_SetPoint := 'True'} : "LAF_InterfaceSignalsBool";
      instSignals41Right { S7_SetPoint := 'True'} : "LAF_InterfaceSignalsBool";
      instSignals42Left { S7_SetPoint := 'True'} : "LAF_InterfaceSignalsBool";
      instSignals42Right { S7_SetPoint := 'True'} : "LAF_InterfaceSignalsBool";
      instSignals43Left { S7_SetPoint := 'True'} : "LAF_InterfaceSignalsBool";
      instSignals43Right { S7_SetPoint := 'True'} : "LAF_InterfaceSignalsBool";
      instSignals44Left { S7_SetPoint := 'True'} : "LAF_InterfaceSignalsBool";
      instSignals44Right { S7_SetPoint := 'True'} : "LAF_InterfaceSignalsBool";
      instSignals45Left { S7_SetPoint := 'True'} : "LAF_InterfaceSignalsBool";
      instSignals45Right { S7_SetPoint := 'True'} : "LAF_InterfaceSignalsBool";
      instSignals46Left { S7_SetPoint := 'True'} : "LAF_InterfaceSignalsBool";
      instSignals46Right { S7_SetPoint := 'True'} : "LAF_InterfaceSignalsBool";
      instSignals47Left { S7_SetPoint := 'True'} : "LAF_InterfaceSignalsBool";
      instSignals47Right { S7_SetPoint := 'True'} : "LAF_InterfaceSignalsBool";
      instSignals48Left { S7_SetPoint := 'True'} : "LAF_InterfaceSignalsBool";
      instSignals48Right { S7_SetPoint := 'True'} : "LAF_InterfaceSignalsBool";
      instSignals49Left { S7_SetPoint := 'True'} : "LAF_InterfaceSignalsBool";
      instSignals49Right { S7_SetPoint := 'True'} : "LAF_InterfaceSignalsBool";
      instSignals50Left { S7_SetPoint := 'True'} : "LAF_InterfaceSignalsBool";
      instSignals50Right { S7_SetPoint := 'True'} : "LAF_InterfaceSignalsBool";
      instSignals51Left { S7_SetPoint := 'True'} : "LAF_InterfaceSignalsBool";
      instSignals51Right { S7_SetPoint := 'True'} : "LAF_InterfaceSignalsBool";
      instSignals52Left { S7_SetPoint := 'True'} : "LAF_InterfaceSignalsBool";
      instSignals52Right { S7_SetPoint := 'True'} : "LAF_InterfaceSignalsBool";
      instSignals53Left { S7_SetPoint := 'True'} : "LAF_InterfaceSignalsBool";
      instSignals53Right { S7_SetPoint := 'True'} : "LAF_InterfaceSignalsBool";
      instSignals54Left { S7_SetPoint := 'True'} : "LAF_InterfaceSignalsBool";
      instSignals54Right { S7_SetPoint := 'True'} : "LAF_InterfaceSignalsBool";
      instSignals55Left { S7_SetPoint := 'True'} : "LAF_InterfaceSignalsBool";
      instSignals55Right { S7_SetPoint := 'True'} : "LAF_InterfaceSignalsBool";
      instSignals56Left { S7_SetPoint := 'True'} : "LAF_InterfaceSignalsBool";
      instSignals56Right { S7_SetPoint := 'True'} : "LAF_InterfaceSignalsBool";
      instSignals57Left { S7_SetPoint := 'True'} : "LAF_InterfaceSignalsBool";
      instSignals57Right { S7_SetPoint := 'True'} : "LAF_InterfaceSignalsBool";
      instSignals58Left { S7_SetPoint := 'True'} : "LAF_InterfaceSignalsBool";
      instSignals58Right { S7_SetPoint := 'True'} : "LAF_InterfaceSignalsBool";
      instSignals59Left { S7_SetPoint := 'True'} : "LAF_InterfaceSignalsBool";
      instSignals59Right { S7_SetPoint := 'True'} : "LAF_InterfaceSignalsBool";
      instSignals60Left { S7_SetPoint := 'True'} : "LAF_InterfaceSignalsBool";
      instSignals60Right { S7_SetPoint := 'True'} : "LAF_InterfaceSignalsBool";
      instSignals61Left { S7_SetPoint := 'True'} : "LAF_InterfaceSignalsBool";
      instSignals61Right { S7_SetPoint := 'True'} : "LAF_InterfaceSignalsBool";
      instSignals62Left { S7_SetPoint := 'True'} : "LAF_InterfaceSignalsBool";
      instSignals62Right { S7_SetPoint := 'True'} : "LAF_InterfaceSignalsBool";
      instSignals63Left { S7_SetPoint := 'True'} : "LAF_InterfaceSignalsBool";
      instSignals63Right { S7_SetPoint := 'True'} : "LAF_InterfaceSignalsBool";
      instSignals64Left { S7_SetPoint := 'True'} : "LAF_InterfaceSignalsBool";
      instSignals64Right { S7_SetPoint := 'True'} : "LAF_InterfaceSignalsBool";
      instSignals65Left { S7_SetPoint := 'True'} : "LAF_InterfaceSignalsBool";
      instSignals65Right { S7_SetPoint := 'True'} : "LAF_InterfaceSignalsBool";
      instSignals66Left { S7_SetPoint := 'True'} : "LAF_InterfaceSignalsBool";
      instSignals66Right { S7_SetPoint := 'True'} : "LAF_InterfaceSignalsBool";
      instSignals67Left { S7_SetPoint := 'True'} : "LAF_InterfaceSignalsBool";
      instSignals67Right { S7_SetPoint := 'True'} : "LAF_InterfaceSignalsBool";
      instSignals68Left { S7_SetPoint := 'True'} : "LAF_InterfaceSignalsBool";
      instSignals68Right { S7_SetPoint := 'True'} : "LAF_InterfaceSignalsBool";
      instSignals69Left { S7_SetPoint := 'True'} : "LAF_InterfaceSignalsBool";
      instSignals69Right { S7_SetPoint := 'True'} : "LAF_InterfaceSignalsBool";
      instSignals70Left { S7_SetPoint := 'True'} : "LAF_InterfaceSignalsBool";
      instSignals70Right { S7_SetPoint := 'True'} : "LAF_InterfaceSignalsBool";
      instSignals71Left { S7_SetPoint := 'True'} : "LAF_InterfaceSignalsBool";
      instSignals71Right { S7_SetPoint := 'True'} : "LAF_InterfaceSignalsBool";
      instSignals72Left { S7_SetPoint := 'True'} : "LAF_InterfaceSignalsBool";
      instSignals72Right { S7_SetPoint := 'True'} : "LAF_InterfaceSignalsBool";
      instSignals73Left { S7_SetPoint := 'True'} : "LAF_InterfaceSignalsBool";
      instSignals73Right { S7_SetPoint := 'True'} : "LAF_InterfaceSignalsBool";
      instSignals74Left { S7_SetPoint := 'True'} : "LAF_InterfaceSignalsBool";
      instSignals74Right { S7_SetPoint := 'True'} : "LAF_InterfaceSignalsBool";
      instSignals75Left { S7_SetPoint := 'True'} : "LAF_InterfaceSignalsBool";
      instSignals75Right { S7_SetPoint := 'True'} : "LAF_InterfaceSignalsBool";
      instSignals76Left { S7_SetPoint := 'True'} : "LAF_InterfaceSignalsBool";
      instSignals76Right { S7_SetPoint := 'True'} : "LAF_InterfaceSignalsBool";
      instSignals77Left { S7_SetPoint := 'True'} : "LAF_InterfaceSignalsBool";
      instSignals77Right { S7_SetPoint := 'True'} : "LAF_InterfaceSignalsBool";
      instSignals78Left { S7_SetPoint := 'True'} : "LAF_InterfaceSignalsBool";
      instSignals78Right { S7_SetPoint := 'True'} : "LAF_InterfaceSignalsBool";
      instSignals79Left { S7_SetPoint := 'True'} : "LAF_InterfaceSignalsBool";
      instSignals79Right { S7_SetPoint := 'True'} : "LAF_InterfaceSignalsBool";
      instSignals80Left { S7_SetPoint := 'True'} : "LAF_InterfaceSignalsBool";
      instSignals80Right { S7_SetPoint := 'True'} : "LAF_InterfaceSignalsBool";
      instSignals81Left { S7_SetPoint := 'True'} : "LAF_InterfaceSignalsBool";
      instSignals81Right { S7_SetPoint := 'True'} : "LAF_InterfaceSignalsBool";
      instSignals82Left { S7_SetPoint := 'True'} : "LAF_InterfaceSignalsBool";
      instSignals82Right { S7_SetPoint := 'True'} : "LAF_InterfaceSignalsBool";
      instSignals83Left { S7_SetPoint := 'True'} : "LAF_InterfaceSignalsBool";
      instSignals83Right { S7_SetPoint := 'True'} : "LAF_InterfaceSignalsBool";
      instSignals84Left { S7_SetPoint := 'True'} : "LAF_InterfaceSignalsBool";
      instSignals84Right { S7_SetPoint := 'True'} : "LAF_InterfaceSignalsBool";
      instSignals85Left { S7_SetPoint := 'True'} : "LAF_InterfaceSignalsBool";
      instSignals85Right { S7_SetPoint := 'True'} : "LAF_InterfaceSignalsBool";
      instSignals86Left { S7_SetPoint := 'True'} : "LAF_InterfaceSignalsBool";
      instSignals86Right { S7_SetPoint := 'True'} : "LAF_InterfaceSignalsBool";
      instSignals87Left { S7_SetPoint := 'True'} : "LAF_InterfaceSignalsBool";
      instSignals87Right { S7_SetPoint := 'True'} : "LAF_InterfaceSignalsBool";
      instSignals88Left { S7_SetPoint := 'True'} : "LAF_InterfaceSignalsBool";
      instSignals88Right { S7_SetPoint := 'True'} : "LAF_InterfaceSignalsBool";
      instSignals89Left { S7_SetPoint := 'True'} : "LAF_InterfaceSignalsBool";
      instSignals89Right { S7_SetPoint := 'True'} : "LAF_InterfaceSignalsBool";
      instSignals90Left { S7_SetPoint := 'True'} : "LAF_InterfaceSignalsBool";
      instSignals90Right { S7_SetPoint := 'True'} : "LAF_InterfaceSignalsBool";
      instSignals91Left { S7_SetPoint := 'True'} : "LAF_InterfaceSignalsBool";
      instSignals91Right { S7_SetPoint := 'True'} : "LAF_InterfaceSignalsBool";
      instSignals92Left { S7_SetPoint := 'True'} : "LAF_InterfaceSignalsBool";
      instSignals92Right { S7_SetPoint := 'True'} : "LAF_InterfaceSignalsBool";
      instSignals93Left { S7_SetPoint := 'True'} : "LAF_InterfaceSignalsBool";
      instSignals93Right { S7_SetPoint := 'True'} : "LAF_InterfaceSignalsBool";
      instSignals94Left { S7_SetPoint := 'True'} : "LAF_InterfaceSignalsBool";
      instSignals94Right { S7_SetPoint := 'True'} : "LAF_InterfaceSignalsBool";
      instSignals95Left { S7_SetPoint := 'True'} : "LAF_InterfaceSignalsBool";
      instSignals95Right { S7_SetPoint := 'True'} : "LAF_InterfaceSignalsBool";
      instSignals96Left { S7_SetPoint := 'True'} : "LAF_InterfaceSignalsBool";
      instSignals96Right { S7_SetPoint := 'True'} : "LAF_InterfaceSignalsBool";
      instSignals97Left { S7_SetPoint := 'True'} : "LAF_InterfaceSignalsBool";
      instSignals97Right { S7_SetPoint := 'True'} : "LAF_InterfaceSignalsBool";
      instSignals98Left { S7_SetPoint := 'True'} : "LAF_InterfaceSignalsBool";
      instSignals98Right { S7_SetPoint := 'True'} : "LAF_InterfaceSignalsBool";
      instSignals99Left { S7_SetPoint := 'True'} : "LAF_InterfaceSignalsBool";
      instSignals99Right { S7_SetPoint := 'True'} : "LAF_InterfaceSignalsBool";
   END_VAR
   VAR_TEMP
      tempLoopCounter : DInt;   // temp. Schleifenzähler / temp. Loop Counter
   END_VAR
   VAR_TEMP   // added for the SCL form of the ladder/FBD networks
      _w1 : Bool;
   END_VAR
BEGIN

REGION Network 1: Beschreibung / BLOCK INFO HEADER
   // **Betriebsart Automatik / Hand**  
   // Der Baustein ist keiner Betriebsart / Betriebsartenbereich zugeordnet.  
   // 
   // **Alarme**  
   // Der Baustein generiert keine Alarme.  
   // 
   // #### PLC-Datentypen  
   // Verwendete PLC-Datentypen für den SPS-Programmbaustein und das zugehörige WinCC-Bild.  
   // 
   // {.pageWidth}
   // ![Image](CallInterfaceSignals/de/image1.PNG)
   //  
   //  
   // #### Bausteinaufrufe 
   // Der Baustein “LSicar_InterfaceSignalsBool“ wird in diesem FB als Multi-Instanz aufgerufen, entspr. nebenstehender beispielhafter Darstellung.  
   // 
   // {.pageWidth}
   // ![Image](CallInterfaceSignals/de/image2.PNG)
   //  
   // Um einen neuen FB aufzurufen, ziehen Sie den FB in ein neues Netzwerk, wählen Sie „Multiinstanz“ aus, vergeben Sie einen Namen und parametrieren Sie den FB-Aufruf.  
   // 
   // {.pageWidth}
   // ![Image](CallInterfaceSignals/de/image3.PNG)
   //  
   //  
   // #### Weitere Hinweise 
   // 
   // #### Updateinfo 
   // 
   // #### Weitere Dokumente 
   // 
   // ![Icon](_Icon/reference.PNG)
   // 
   // ..\Library Types\LSicar_InterfaceSignalsBool.pdf
   // SIEMENS AG / (c)Copyright 2023
   // ------------------------------------------------------------------------------
   // Title:            CallInterfaceSignals (FB38)
   // Comment/Function: The block serves as a calling interface of the block “InterfaceSignalsBool“. The block is designed as function block in order to implement the block calls as multi-instances. 
   // Library/Family:   Diag
   // Author:           SICAR
   // Tested with:      ---
   // Engineering:      TIA Portal V19
   // Restrictions:     -
   // Requirements:     ---
   // ------------------------------------------------------------------------------
   // Change log table:
   // Version  | Date       | Expert in charge       | Changes applied
   // ---------|------------|------------------------|------------------------------
   // 01.00.00 | 11.12.2023 | SICAR
   //                         First released version
END_REGION

REGION Network 2: DESCRIPTION
   // Function block and corresponding WinCC screen are prepared for 16 data sets (“InterfaceSignals01“ through .”InterfaceSignals16“) with 32 Boolean signals each.  
   // 
   // **PLC-Data types**   
   // 
   // * LSicar_typeInterfaceSignalsBool 
   // * LSicar _typeInterfaceSignals 
   // * typeInterfaceSignalsHmi 
   // 
   // **WinCC-Faceplate**  
   // 
   // <None> 
   // 
   // **WinCC Diagnostic screen**   
   // 
   // See: ..\Library Types\LSicar_InterfaceSignalsBool.pdf  
   // 
   // **Block call example** 
   // 
   // View in ladder-logic (LAD), without parameter settings.  
   // An executable program call is available in the “SICAR-Startup” project.  
   // 
   // **Calling interface**  
   // 
   // The block is be called once in the cyclic program.  
   // 
   // **Internally used „Extended instructions / blocks“**  
   // 
   // See: ..\Library Types\LSicar_InterfaceSignalsBool.pdf
END_REGION

REGION Network 3: Initialisierung Loop_1 / Initialization Loop_1
   // Vorbesetzen des Schleifenindex / Preset the loop index
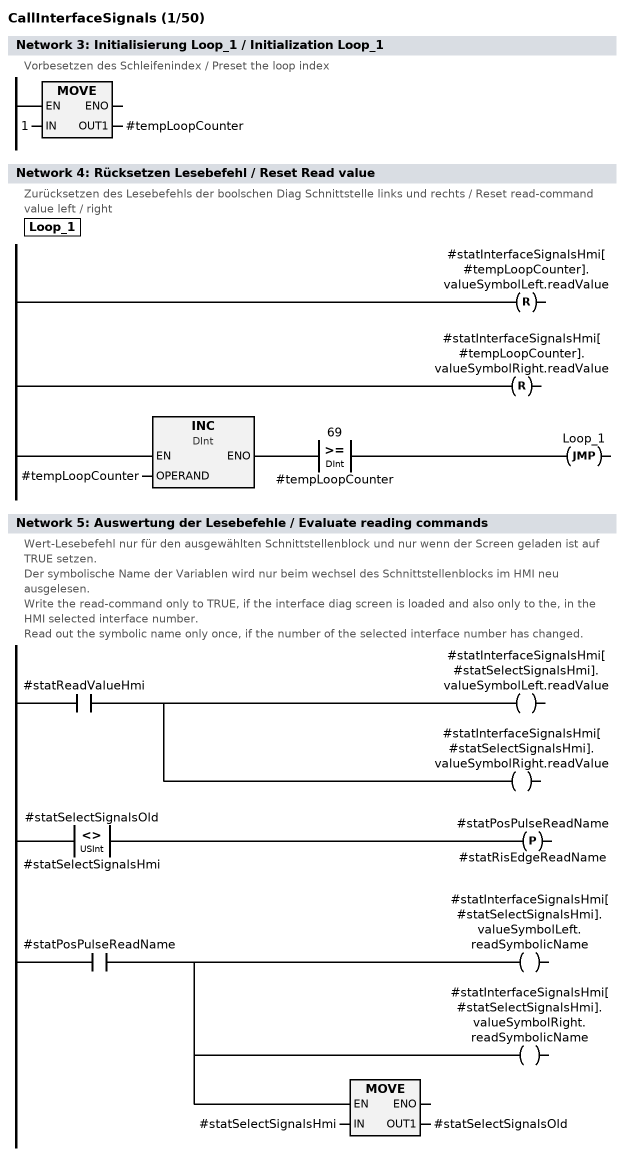
   RUNG wire#powerrail
      Move(in := 1, out1 => #tempLoopCounter)
   END_RUNG
   // the same network as SCL:
   #tempLoopCounter := 1;
END_REGION

REGION Network 4: Rücksetzen Lesebefehl / Reset Read value
   // Zurücksetzen des Lesebefehls der boolschen Diag Schnittstelle links und rechts / Reset read-command value left / right
   Label( Loop_1 )
   RUNG wire#powerrail
      R_Coil( #statInterfaceSignalsHmi[#tempLoopCounter].valueSymbolLeft.readValue )
   END_RUNG
   RUNG wire#powerrail
      R_Coil( #statInterfaceSignalsHmi[#tempLoopCounter].valueSymbolRight.readValue )
   END_RUNG
   RUNG wire#powerrail
      { S7_Templates := "DestType := DInt" } Inc( #tempLoopCounter )
      { S7_Templates := "SrcType := DInt" } GE_Contact(in1 := 69, in2 := #tempLoopCounter)
      JumpCoil( Loop_1 )
   END_RUNG
   // the same network as SCL:
   Loop_1:
   #statInterfaceSignalsHmi[#tempLoopCounter].valueSymbolLeft.readValue := FALSE;
   #statInterfaceSignalsHmi[#tempLoopCounter].valueSymbolRight.readValue := FALSE;
   #tempLoopCounter := #tempLoopCounter + 1;
   IF 69 >= #tempLoopCounter THEN GOTO Loop_1; END_IF;
END_REGION

REGION Network 5: Auswertung der Lesebefehle / Evaluate reading commands
   // Wert-Lesebefehl nur für den ausgewählten Schnittstellenblock und nur wenn der Screen geladen ist auf TRUE setzen.
   // Der symbolische Name der Variablen wird nur beim wechsel des Schnittstellenblocks im HMI neu ausgelesen.
   // Write the read-command only to TRUE, if the interface diag screen is loaded and also only to the, in the HMI selected interface number.
   // Read out the symbolic name only once, if the number of the selected interface number has changed.
   #statInterfaceSignalsHmi[#statSelectSignalsHmi].valueSymbolLeft.readValue := #statReadValueHmi;
   #statInterfaceSignalsHmi[#statSelectSignalsHmi].valueSymbolRight.readValue := #statReadValueHmi;
   #_w1 := #statSelectSignalsOld <> #statSelectSignalsHmi;
   #statPosPulseReadName := #_w1 AND NOT #statRisEdgeReadName;   // rising edge
   #statRisEdgeReadName := #_w1;
   #statInterfaceSignalsHmi[#statSelectSignalsHmi].valueSymbolLeft.readSymbolicName := #statPosPulseReadName;
   #statInterfaceSignalsHmi[#statSelectSignalsHmi].valueSymbolRight.readSymbolicName := #statPosPulseReadName;
   IF #statPosPulseReadName THEN #statSelectSignalsOld := #statSelectSignalsHmi; END_IF;
END_REGION

REGION Network 6: Interface Signals 03 -Example: System flags & Clock flags- / Interface Signals 01
   // Aufruf des Schnittstellen Signal Bausteins für die Systemvariablen / Call the interface signals bool blocks of system tags
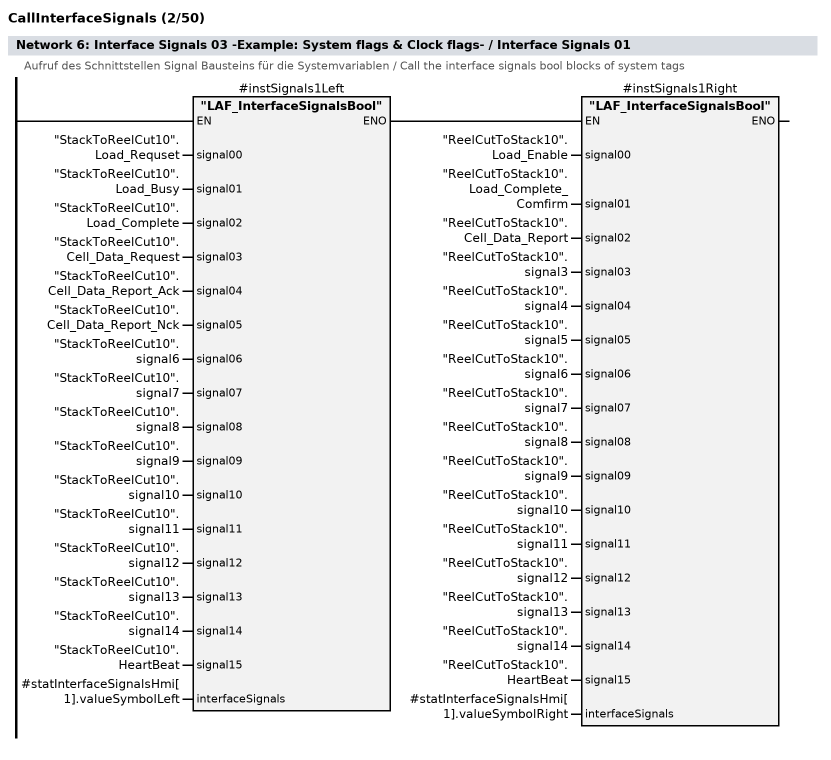
   RUNG wire#powerrail
      #instSignals1Left(signal00 := "StackToReelCut10".Load_Requset, signal01 := "StackToReelCut10".Load_Busy, signal02 := "StackToReelCut10".Load_Complete, signal03 := "StackToReelCut10".Cell_Data_Request, signal04 := "StackToReelCut10".Cell_Data_Report_Ack, signal05 := "StackToReelCut10".Cell_Data_Report_Nck, signal06 := "StackToReelCut10".signal6, signal07 := "StackToReelCut10".signal7, signal08 := "StackToReelCut10".signal8, signal09 := "StackToReelCut10".signal9, signal10 := "StackToReelCut10".signal10, signal11 := "StackToReelCut10".signal11, signal12 := "StackToReelCut10".signal12, signal13 := "StackToReelCut10".signal13, signal14 := "StackToReelCut10".signal14, signal15 := "StackToReelCut10".HeartBeat, interfaceSignals := #statInterfaceSignalsHmi[1].valueSymbolLeft)
      #instSignals1Right(signal00 := "ReelCutToStack10".Load_Enable, signal01 := "ReelCutToStack10".Load_Complete_Comfirm, signal02 := "ReelCutToStack10".Cell_Data_Report, signal03 := "ReelCutToStack10".signal3, signal04 := "ReelCutToStack10".signal4, signal05 := "ReelCutToStack10".signal5, signal06 := "ReelCutToStack10".signal6, signal07 := "ReelCutToStack10".signal7, signal08 := "ReelCutToStack10".signal8, signal09 := "ReelCutToStack10".signal9, signal10 := "ReelCutToStack10".signal10, signal11 := "ReelCutToStack10".signal11, signal12 := "ReelCutToStack10".signal12, signal13 := "ReelCutToStack10".signal13, signal14 := "ReelCutToStack10".signal14, signal15 := "ReelCutToStack10".HeartBeat, interfaceSignals := #statInterfaceSignalsHmi[1].valueSymbolRight)
   END_RUNG
   // the same network as SCL:
   #instSignals1Left(signal00 := "StackToReelCut10".Load_Requset,   // "LAF_InterfaceSignalsBool"
                     signal01 := "StackToReelCut10".Load_Busy,
                     signal02 := "StackToReelCut10".Load_Complete,
                     signal03 := "StackToReelCut10".Cell_Data_Request,
                     signal04 := "StackToReelCut10".Cell_Data_Report_Ack,
                     signal05 := "StackToReelCut10".Cell_Data_Report_Nck,
                     signal06 := "StackToReelCut10".signal6,
                     signal07 := "StackToReelCut10".signal7,
                     signal08 := "StackToReelCut10".signal8,
                     signal09 := "StackToReelCut10".signal9,
                     signal10 := "StackToReelCut10".signal10,
                     signal11 := "StackToReelCut10".signal11,
                     signal12 := "StackToReelCut10".signal12,
                     signal13 := "StackToReelCut10".signal13,
                     signal14 := "StackToReelCut10".signal14,
                     signal15 := "StackToReelCut10".HeartBeat,
                     interfaceSignals := #statInterfaceSignalsHmi[1].valueSymbolLeft,
                     ENO => #_w1);
   IF #_w1 THEN
       #instSignals1Right(signal00 := "ReelCutToStack10".Load_Enable,   // "LAF_InterfaceSignalsBool"
                          signal01 := "ReelCutToStack10".Load_Complete_Comfirm,
                          signal02 := "ReelCutToStack10".Cell_Data_Report,
                          signal03 := "ReelCutToStack10".signal3,
                          signal04 := "ReelCutToStack10".signal4,
                          signal05 := "ReelCutToStack10".signal5,
                          signal06 := "ReelCutToStack10".signal6,
                          signal07 := "ReelCutToStack10".signal7,
                          signal08 := "ReelCutToStack10".signal8,
                          signal09 := "ReelCutToStack10".signal9,
                          signal10 := "ReelCutToStack10".signal10,
                          signal11 := "ReelCutToStack10".signal11,
                          signal12 := "ReelCutToStack10".signal12,
                          signal13 := "ReelCutToStack10".signal13,
                          signal14 := "ReelCutToStack10".signal14,
                          signal15 := "ReelCutToStack10".HeartBeat,
                          interfaceSignals := #statInterfaceSignalsHmi[1].valueSymbolRight);
   END_IF;
END_REGION

REGION Network 7: Interface Signals 03 -Example: System flags & Clock flags- / Interface Signals 02
   // Aufruf des Schnittstellen Signal Bausteins für die Systemvariablen / Call the interface signals bool blocks of system tags
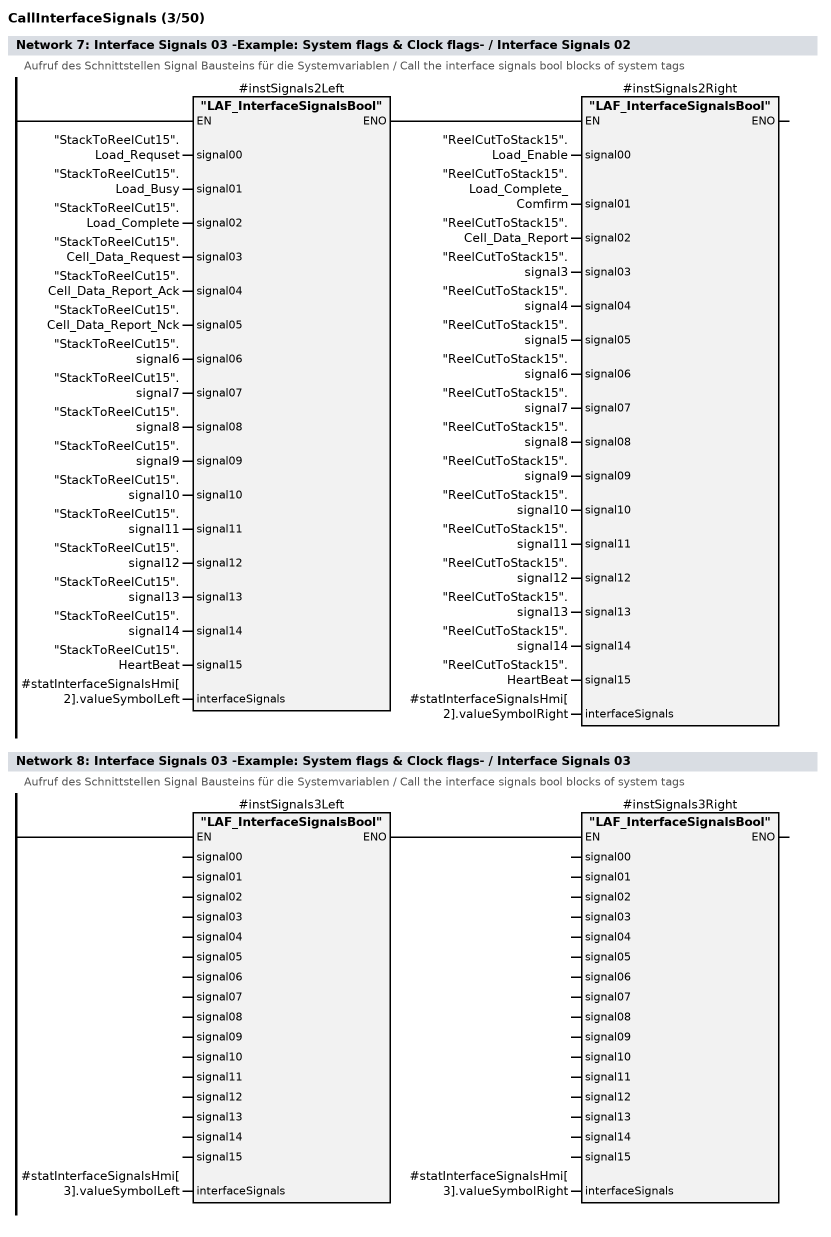
   RUNG wire#powerrail
      #instSignals2Left(signal00 := "StackToReelCut15".Load_Requset, signal01 := "StackToReelCut15".Load_Busy, signal02 := "StackToReelCut15".Load_Complete, signal03 := "StackToReelCut15".Cell_Data_Request, signal04 := "StackToReelCut15".Cell_Data_Report_Ack, signal05 := "StackToReelCut15".Cell_Data_Report_Nck, signal06 := "StackToReelCut15".signal6, signal07 := "StackToReelCut15".signal7, signal08 := "StackToReelCut15".signal8, signal09 := "StackToReelCut15".signal9, signal10 := "StackToReelCut15".signal10, signal11 := "StackToReelCut15".signal11, signal12 := "StackToReelCut15".signal12, signal13 := "StackToReelCut15".signal13, signal14 := "StackToReelCut15".signal14, signal15 := "StackToReelCut15".HeartBeat, interfaceSignals := #statInterfaceSignalsHmi[2].valueSymbolLeft)
      #instSignals2Right(signal00 := "ReelCutToStack15".Load_Enable, signal01 := "ReelCutToStack15".Load_Complete_Comfirm, signal02 := "ReelCutToStack15".Cell_Data_Report, signal03 := "ReelCutToStack15".signal3, signal04 := "ReelCutToStack15".signal4, signal05 := "ReelCutToStack15".signal5, signal06 := "ReelCutToStack15".signal6, signal07 := "ReelCutToStack15".signal7, signal08 := "ReelCutToStack15".signal8, signal09 := "ReelCutToStack15".signal9, signal10 := "ReelCutToStack15".signal10, signal11 := "ReelCutToStack15".signal11, signal12 := "ReelCutToStack15".signal12, signal13 := "ReelCutToStack15".signal13, signal14 := "ReelCutToStack15".signal14, signal15 := "ReelCutToStack15".HeartBeat, interfaceSignals := #statInterfaceSignalsHmi[2].valueSymbolRight)
   END_RUNG
   // the same network as SCL:
   #instSignals2Left(signal00 := "StackToReelCut15".Load_Requset,   // "LAF_InterfaceSignalsBool"
                     signal01 := "StackToReelCut15".Load_Busy,
                     signal02 := "StackToReelCut15".Load_Complete,
                     signal03 := "StackToReelCut15".Cell_Data_Request,
                     signal04 := "StackToReelCut15".Cell_Data_Report_Ack,
                     signal05 := "StackToReelCut15".Cell_Data_Report_Nck,
                     signal06 := "StackToReelCut15".signal6,
                     signal07 := "StackToReelCut15".signal7,
                     signal08 := "StackToReelCut15".signal8,
                     signal09 := "StackToReelCut15".signal9,
                     signal10 := "StackToReelCut15".signal10,
                     signal11 := "StackToReelCut15".signal11,
                     signal12 := "StackToReelCut15".signal12,
                     signal13 := "StackToReelCut15".signal13,
                     signal14 := "StackToReelCut15".signal14,
                     signal15 := "StackToReelCut15".HeartBeat,
                     interfaceSignals := #statInterfaceSignalsHmi[2].valueSymbolLeft,
                     ENO => #_w1);
   IF #_w1 THEN
       #instSignals2Right(signal00 := "ReelCutToStack15".Load_Enable,   // "LAF_InterfaceSignalsBool"
                          signal01 := "ReelCutToStack15".Load_Complete_Comfirm,
                          signal02 := "ReelCutToStack15".Cell_Data_Report,
                          signal03 := "ReelCutToStack15".signal3,
                          signal04 := "ReelCutToStack15".signal4,
                          signal05 := "ReelCutToStack15".signal5,
                          signal06 := "ReelCutToStack15".signal6,
                          signal07 := "ReelCutToStack15".signal7,
                          signal08 := "ReelCutToStack15".signal8,
                          signal09 := "ReelCutToStack15".signal9,
                          signal10 := "ReelCutToStack15".signal10,
                          signal11 := "ReelCutToStack15".signal11,
                          signal12 := "ReelCutToStack15".signal12,
                          signal13 := "ReelCutToStack15".signal13,
                          signal14 := "ReelCutToStack15".signal14,
                          signal15 := "ReelCutToStack15".HeartBeat,
                          interfaceSignals := #statInterfaceSignalsHmi[2].valueSymbolRight);
   END_IF;
END_REGION

REGION Network 8: Interface Signals 03 -Example: System flags & Clock flags- / Interface Signals 03
   // Aufruf des Schnittstellen Signal Bausteins für die Systemvariablen / Call the interface signals bool blocks of system tags
   RUNG wire#powerrail
      #instSignals3Left(signal00 :=, signal01 :=, signal02 :=, signal03 :=, signal04 :=, signal05 :=, signal06 :=, signal07 :=, signal08 :=, signal09 :=, signal10 :=, signal11 :=, signal12 :=, signal13 :=, signal14 :=, signal15 :=, interfaceSignals := #statInterfaceSignalsHmi[3].valueSymbolLeft)
      #instSignals3Right(signal00 :=, signal01 :=, signal02 :=, signal03 :=, signal04 :=, signal05 :=, signal06 :=, signal07 :=, signal08 :=, signal09 :=, signal10 :=, signal11 :=, signal12 :=, signal13 :=, signal14 :=, signal15 :=, interfaceSignals := #statInterfaceSignalsHmi[3].valueSymbolRight)
   END_RUNG
   // the same network as SCL:
   #instSignals3Left(interfaceSignals := #statInterfaceSignalsHmi[3].valueSymbolLeft, ENO => #_w1);   // "LAF_InterfaceSignalsBool"
   IF #_w1 THEN
       #instSignals3Right(interfaceSignals := #statInterfaceSignalsHmi[3].valueSymbolRight);   // "LAF_InterfaceSignalsBool"
   END_IF;
END_REGION

REGION Network 9: Interface Signals 04 -Example: Model Flex-Pro-Line - IN/OUT- / Interface Signals 04
   // Aufruf des Schnittstellen Signal Bausteins Ba-Bereich 4 / Call the interface signals bool blocks of opmode 4
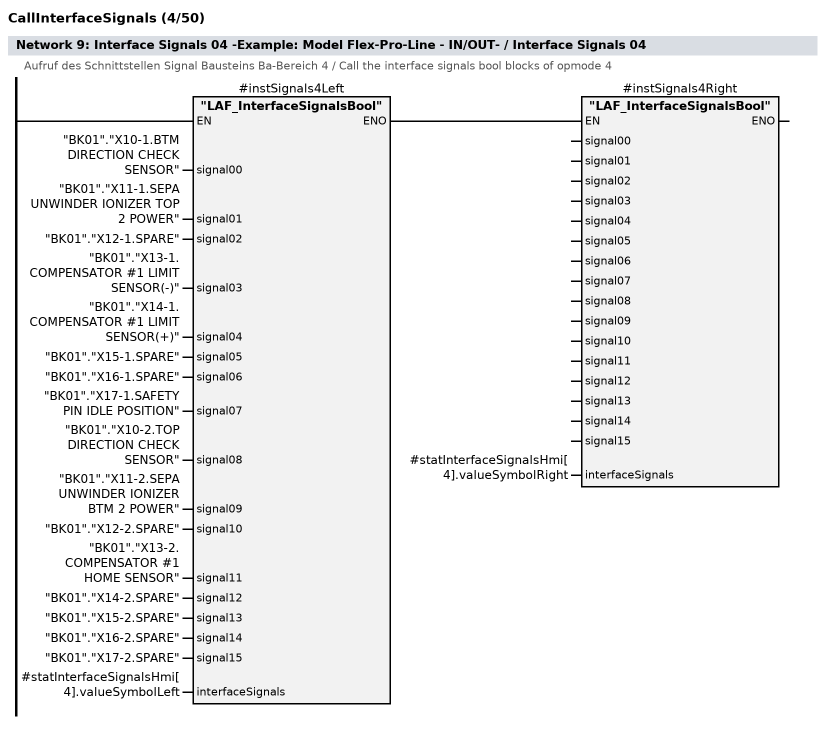
   RUNG wire#powerrail
      #instSignals4Left(signal00 := "BK01"."X10-1.BTM DIRECTION CHECK SENSOR", signal01 := "BK01"."X11-1.SEPA UNWINDER IONIZER TOP 2 POWER", signal02 := "BK01"."X12-1.SPARE", signal03 := "BK01"."X13-1.COMPENSATOR #1 LIMIT SENSOR(-)", signal04 := "BK01"."X14-1.COMPENSATOR #1 LIMIT SENSOR(+)", signal05 := "BK01"."X15-1.SPARE", signal06 := "BK01"."X16-1.SPARE", signal07 := "BK01"."X17-1.SAFETY PIN IDLE POSITION", signal08 := "BK01"."X10-2.TOP DIRECTION CHECK SENSOR", signal09 := "BK01"."X11-2.SEPA UNWINDER IONIZER BTM 2 POWER", signal10 := "BK01"."X12-2.SPARE", signal11 := "BK01"."X13-2.COMPENSATOR #1 HOME SENSOR", signal12 := "BK01"."X14-2.SPARE", signal13 := "BK01"."X15-2.SPARE", signal14 := "BK01"."X16-2.SPARE", signal15 := "BK01"."X17-2.SPARE", interfaceSignals := #statInterfaceSignalsHmi[4].valueSymbolLeft)
      #instSignals4Right(signal00 :=, signal01 :=, signal02 :=, signal03 :=, signal04 :=, signal05 :=, signal06 :=, signal07 :=, signal08 :=, signal09 :=, signal10 :=, signal11 :=, signal12 :=, signal13 :=, signal14 :=, signal15 :=, interfaceSignals := #statInterfaceSignalsHmi[4].valueSymbolRight)
   END_RUNG
   // the same network as SCL:
   #instSignals4Left(signal00 := "BK01"."X10-1.BTM DIRECTION CHECK SENSOR",   // "LAF_InterfaceSignalsBool"
                     signal01 := "BK01"."X11-1.SEPA UNWINDER IONIZER TOP 2 POWER",
                     signal02 := "BK01"."X12-1.SPARE",
                     signal03 := "BK01"."X13-1.COMPENSATOR #1 LIMIT SENSOR(-)",
                     signal04 := "BK01"."X14-1.COMPENSATOR #1 LIMIT SENSOR(+)",
                     signal05 := "BK01"."X15-1.SPARE",
                     signal06 := "BK01"."X16-1.SPARE",
                     signal07 := "BK01"."X17-1.SAFETY PIN IDLE POSITION",
                     signal08 := "BK01"."X10-2.TOP DIRECTION CHECK SENSOR",
                     signal09 := "BK01"."X11-2.SEPA UNWINDER IONIZER BTM 2 POWER",
                     signal10 := "BK01"."X12-2.SPARE",
                     signal11 := "BK01"."X13-2.COMPENSATOR #1 HOME SENSOR",
                     signal12 := "BK01"."X14-2.SPARE",
                     signal13 := "BK01"."X15-2.SPARE",
                     signal14 := "BK01"."X16-2.SPARE",
                     signal15 := "BK01"."X17-2.SPARE",
                     interfaceSignals := #statInterfaceSignalsHmi[4].valueSymbolLeft,
                     ENO => #_w1);
   IF #_w1 THEN
       #instSignals4Right(interfaceSignals := #statInterfaceSignalsHmi[4].valueSymbolRight);   // "LAF_InterfaceSignalsBool"
   END_IF;
END_REGION

REGION Network 10: Interface Signals 05 -Example: Model Flex-Pro-Line - IN/OUT- / Interface Signals 05
   // Aufruf des Schnittstellen Signal Bausteins Ba-Bereich 4 / Call the interface signals bool blocks of opmode 4
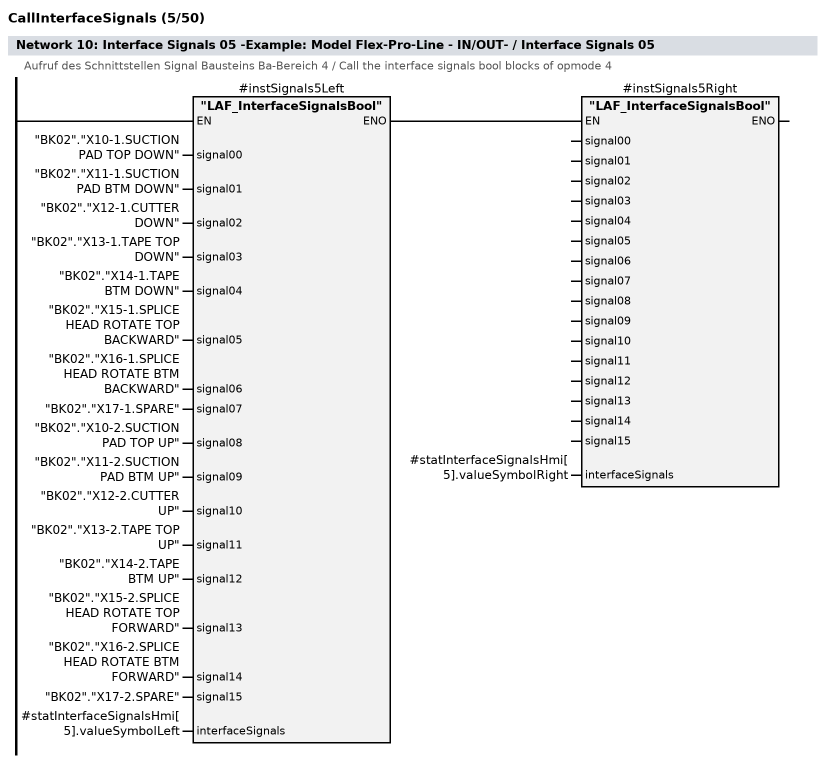
   RUNG wire#powerrail
      #instSignals5Left(signal00 := "BK02"."X10-1.SUCTION PAD TOP DOWN", signal01 := "BK02"."X11-1.SUCTION PAD BTM DOWN", signal02 := "BK02"."X12-1.CUTTER DOWN", signal03 := "BK02"."X13-1.TAPE TOP DOWN", signal04 := "BK02"."X14-1.TAPE BTM DOWN", signal05 := "BK02"."X15-1.SPLICE HEAD ROTATE TOP BACKWARD", signal06 := "BK02"."X16-1.SPLICE HEAD ROTATE BTM BACKWARD", signal07 := "BK02"."X17-1.SPARE", signal08 := "BK02"."X10-2.SUCTION PAD TOP UP", signal09 := "BK02"."X11-2.SUCTION PAD BTM UP", signal10 := "BK02"."X12-2.CUTTER UP", signal11 := "BK02"."X13-2.TAPE TOP UP", signal12 := "BK02"."X14-2.TAPE BTM UP", signal13 := "BK02"."X15-2.SPLICE HEAD ROTATE TOP FORWARD", signal14 := "BK02"."X16-2.SPLICE HEAD ROTATE BTM FORWARD", signal15 := "BK02"."X17-2.SPARE", interfaceSignals := #statInterfaceSignalsHmi[5].valueSymbolLeft)
      #instSignals5Right(signal00 :=, signal01 :=, signal02 :=, signal03 :=, signal04 :=, signal05 :=, signal06 :=, signal07 :=, signal08 :=, signal09 :=, signal10 :=, signal11 :=, signal12 :=, signal13 :=, signal14 :=, signal15 :=, interfaceSignals := #statInterfaceSignalsHmi[5].valueSymbolRight)
   END_RUNG
   // the same network as SCL:
   #instSignals5Left(signal00 := "BK02"."X10-1.SUCTION PAD TOP DOWN",   // "LAF_InterfaceSignalsBool"
                     signal01 := "BK02"."X11-1.SUCTION PAD BTM DOWN",
                     signal02 := "BK02"."X12-1.CUTTER DOWN",
                     signal03 := "BK02"."X13-1.TAPE TOP DOWN",
                     signal04 := "BK02"."X14-1.TAPE BTM DOWN",
                     signal05 := "BK02"."X15-1.SPLICE HEAD ROTATE TOP BACKWARD",
                     signal06 := "BK02"."X16-1.SPLICE HEAD ROTATE BTM BACKWARD",
                     signal07 := "BK02"."X17-1.SPARE",
                     signal08 := "BK02"."X10-2.SUCTION PAD TOP UP",
                     signal09 := "BK02"."X11-2.SUCTION PAD BTM UP",
                     signal10 := "BK02"."X12-2.CUTTER UP",
                     signal11 := "BK02"."X13-2.TAPE TOP UP",
                     signal12 := "BK02"."X14-2.TAPE BTM UP",
                     signal13 := "BK02"."X15-2.SPLICE HEAD ROTATE TOP FORWARD",
                     signal14 := "BK02"."X16-2.SPLICE HEAD ROTATE BTM FORWARD",
                     signal15 := "BK02"."X17-2.SPARE",
                     interfaceSignals := #statInterfaceSignalsHmi[5].valueSymbolLeft,
                     ENO => #_w1);
   IF #_w1 THEN
       #instSignals5Right(interfaceSignals := #statInterfaceSignalsHmi[5].valueSymbolRight);   // "LAF_InterfaceSignalsBool"
   END_IF;
END_REGION

REGION Network 11: Interface Signals 05 -Example: Model Flex-Pro-Line - IN/OUT- / Interface Signals 06
   // Aufruf des Schnittstellen Signal Bausteins Ba-Bereich 4 / Call the interface signals bool blocks of opmode 4
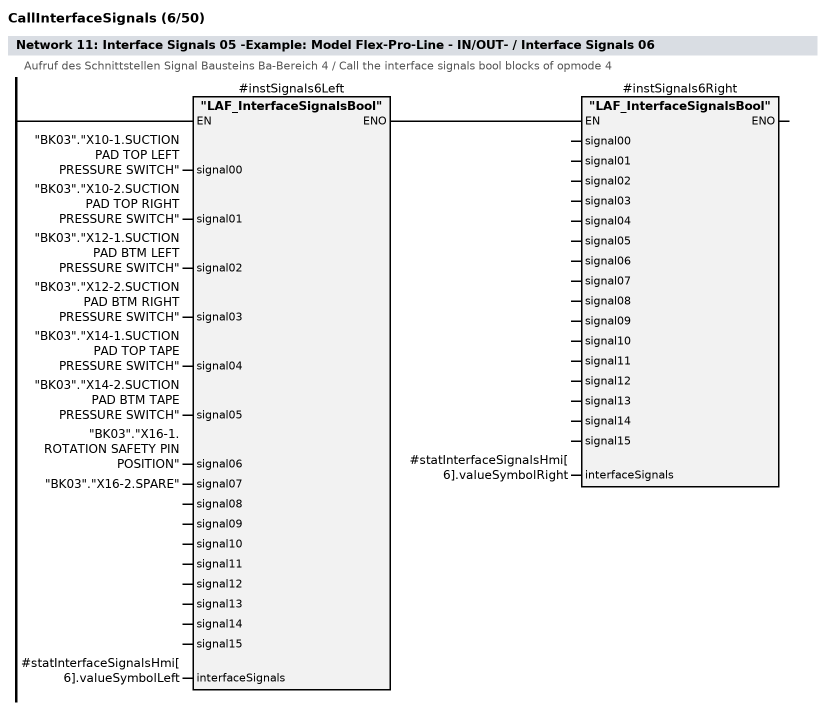
   RUNG wire#powerrail
      #instSignals6Left(signal00 := "BK03"."X10-1.SUCTION PAD TOP LEFT PRESSURE SWITCH", signal01 := "BK03"."X10-2.SUCTION PAD TOP RIGHT PRESSURE SWITCH", signal02 := "BK03"."X12-1.SUCTION PAD BTM LEFT PRESSURE SWITCH", signal03 := "BK03"."X12-2.SUCTION PAD BTM RIGHT PRESSURE SWITCH", signal04 := "BK03"."X14-1.SUCTION PAD TOP TAPE PRESSURE SWITCH", signal05 := "BK03"."X14-2.SUCTION PAD BTM TAPE PRESSURE SWITCH", signal06 := "BK03"."X16-1.ROTATION SAFETY PIN POSITION", signal07 := "BK03"."X16-2.SPARE", signal08 :=, signal09 :=, signal10 :=, signal11 :=, signal12 :=, signal13 :=, signal14 :=, signal15 :=, interfaceSignals := #statInterfaceSignalsHmi[6].valueSymbolLeft)
      #instSignals6Right(signal00 :=, signal01 :=, signal02 :=, signal03 :=, signal04 :=, signal05 :=, signal06 :=, signal07 :=, signal08 :=, signal09 :=, signal10 :=, signal11 :=, signal12 :=, signal13 :=, signal14 :=, signal15 :=, interfaceSignals := #statInterfaceSignalsHmi[6].valueSymbolRight)
   END_RUNG
   // the same network as SCL:
   #instSignals6Left(signal00 := "BK03"."X10-1.SUCTION PAD TOP LEFT PRESSURE SWITCH",   // "LAF_InterfaceSignalsBool"
                     signal01 := "BK03"."X10-2.SUCTION PAD TOP RIGHT PRESSURE SWITCH",
                     signal02 := "BK03"."X12-1.SUCTION PAD BTM LEFT PRESSURE SWITCH",
                     signal03 := "BK03"."X12-2.SUCTION PAD BTM RIGHT PRESSURE SWITCH",
                     signal04 := "BK03"."X14-1.SUCTION PAD TOP TAPE PRESSURE SWITCH",
                     signal05 := "BK03"."X14-2.SUCTION PAD BTM TAPE PRESSURE SWITCH",
                     signal06 := "BK03"."X16-1.ROTATION SAFETY PIN POSITION",
                     signal07 := "BK03"."X16-2.SPARE",
                     interfaceSignals := #statInterfaceSignalsHmi[6].valueSymbolLeft,
                     ENO => #_w1);
   IF #_w1 THEN
       #instSignals6Right(interfaceSignals := #statInterfaceSignalsHmi[6].valueSymbolRight);   // "LAF_InterfaceSignalsBool"
   END_IF;
END_REGION

REGION Network 12: Interface Signals 05 -Example: Model Flex-Pro-Line - IN/OUT- / Interface Signals 07
   // Aufruf des Schnittstellen Signal Bausteins Ba-Bereich 4 / Call the interface signals bool blocks of opmode 4
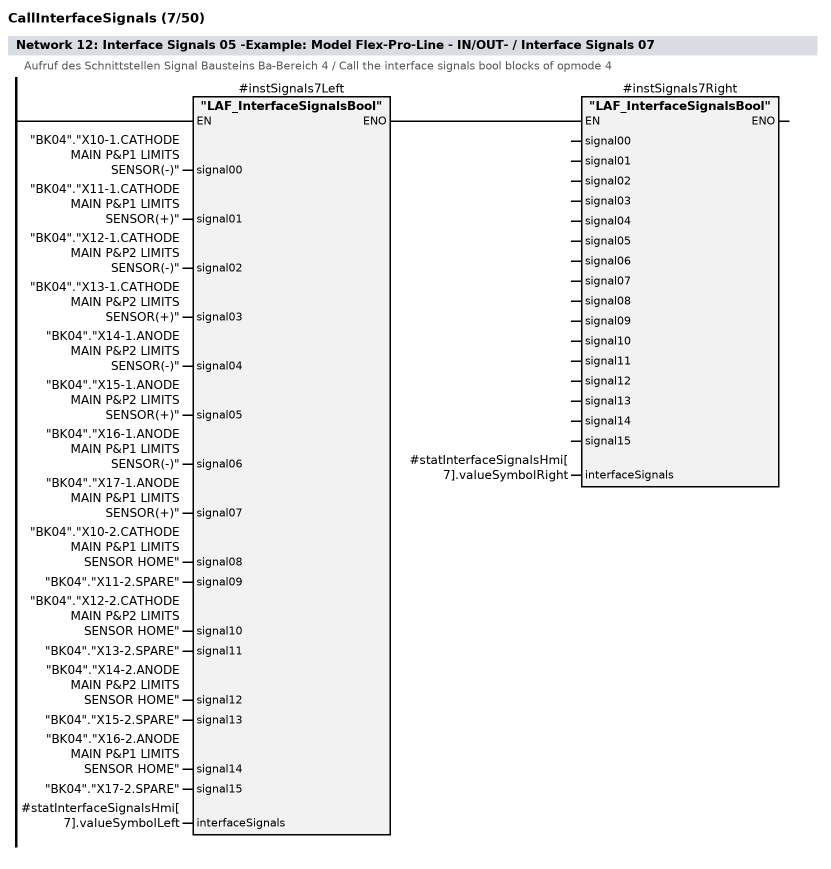
   RUNG wire#powerrail
      #instSignals7Left(signal00 := "BK04"."X10-1.CATHODE MAIN P&P1 LIMITS SENSOR(-)", signal01 := "BK04"."X11-1.CATHODE MAIN P&P1 LIMITS SENSOR(+)", signal02 := "BK04"."X12-1.CATHODE MAIN P&P2 LIMITS SENSOR(-)", signal03 := "BK04"."X13-1.CATHODE MAIN P&P2 LIMITS SENSOR(+)", signal04 := "BK04"."X14-1.ANODE MAIN P&P2 LIMITS SENSOR(-)", signal05 := "BK04"."X15-1.ANODE MAIN P&P2 LIMITS SENSOR(+)", signal06 := "BK04"."X16-1.ANODE MAIN P&P1 LIMITS SENSOR(-)", signal07 := "BK04"."X17-1.ANODE MAIN P&P1 LIMITS SENSOR(+)", signal08 := "BK04"."X10-2.CATHODE MAIN P&P1 LIMITS SENSOR HOME", signal09 := "BK04"."X11-2.SPARE", signal10 := "BK04"."X12-2.CATHODE MAIN P&P2 LIMITS SENSOR HOME", signal11 := "BK04"."X13-2.SPARE", signal12 := "BK04"."X14-2.ANODE MAIN P&P2 LIMITS SENSOR HOME", signal13 := "BK04"."X15-2.SPARE", signal14 := "BK04"."X16-2.ANODE MAIN P&P1 LIMITS SENSOR HOME", signal15 := "BK04"."X17-2.SPARE", interfaceSignals := #statInterfaceSignalsHmi[7].valueSymbolLeft)
      #instSignals7Right(signal00 :=, signal01 :=, signal02 :=, signal03 :=, signal04 :=, signal05 :=, signal06 :=, signal07 :=, signal08 :=, signal09 :=, signal10 :=, signal11 :=, signal12 :=, signal13 :=, signal14 :=, signal15 :=, interfaceSignals := #statInterfaceSignalsHmi[7].valueSymbolRight)
   END_RUNG
   // the same network as SCL:
   #instSignals7Left(signal00 := "BK04"."X10-1.CATHODE MAIN P&P1 LIMITS SENSOR(-)",   // "LAF_InterfaceSignalsBool"
                     signal01 := "BK04"."X11-1.CATHODE MAIN P&P1 LIMITS SENSOR(+)",
                     signal02 := "BK04"."X12-1.CATHODE MAIN P&P2 LIMITS SENSOR(-)",
                     signal03 := "BK04"."X13-1.CATHODE MAIN P&P2 LIMITS SENSOR(+)",
                     signal04 := "BK04"."X14-1.ANODE MAIN P&P2 LIMITS SENSOR(-)",
                     signal05 := "BK04"."X15-1.ANODE MAIN P&P2 LIMITS SENSOR(+)",
                     signal06 := "BK04"."X16-1.ANODE MAIN P&P1 LIMITS SENSOR(-)",
                     signal07 := "BK04"."X17-1.ANODE MAIN P&P1 LIMITS SENSOR(+)",
                     signal08 := "BK04"."X10-2.CATHODE MAIN P&P1 LIMITS SENSOR HOME",
                     signal09 := "BK04"."X11-2.SPARE",
                     signal10 := "BK04"."X12-2.CATHODE MAIN P&P2 LIMITS SENSOR HOME",
                     signal11 := "BK04"."X13-2.SPARE",
                     signal12 := "BK04"."X14-2.ANODE MAIN P&P2 LIMITS SENSOR HOME",
                     signal13 := "BK04"."X15-2.SPARE",
                     signal14 := "BK04"."X16-2.ANODE MAIN P&P1 LIMITS SENSOR HOME",
                     signal15 := "BK04"."X17-2.SPARE",
                     interfaceSignals := #statInterfaceSignalsHmi[7].valueSymbolLeft,
                     ENO => #_w1);
   IF #_w1 THEN
       #instSignals7Right(interfaceSignals := #statInterfaceSignalsHmi[7].valueSymbolRight);   // "LAF_InterfaceSignalsBool"
   END_IF;
END_REGION

REGION Network 13: Interface Signals 05 -Example: Model Flex-Pro-Line - IN/OUT- / Interface Signals 08
   // Aufruf des Schnittstellen Signal Bausteins Ba-Bereich 4 / Call the interface signals bool blocks of opmode 4
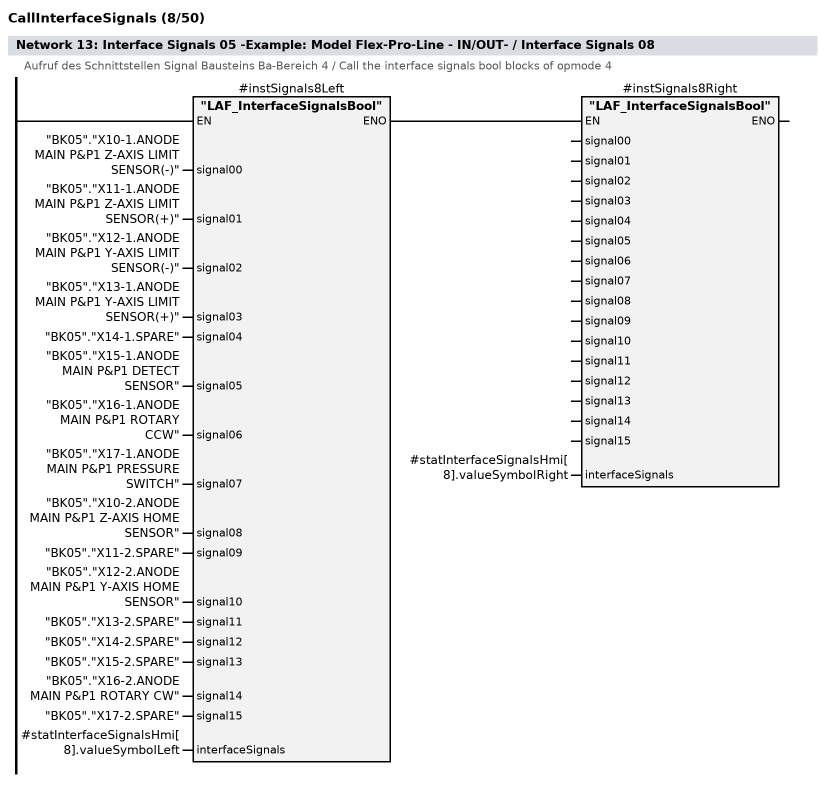
   RUNG wire#powerrail
      #instSignals8Left(signal00 := "BK05"."X10-1.ANODE MAIN P&P1 Z-AXIS LIMIT SENSOR(-)", signal01 := "BK05"."X11-1.ANODE MAIN P&P1 Z-AXIS LIMIT SENSOR(+)", signal02 := "BK05"."X12-1.ANODE MAIN P&P1 Y-AXIS LIMIT SENSOR(-)", signal03 := "BK05"."X13-1.ANODE MAIN P&P1 Y-AXIS LIMIT SENSOR(+)", signal04 := "BK05"."X14-1.SPARE", signal05 := "BK05"."X15-1.ANODE MAIN P&P1 DETECT SENSOR", signal06 := "BK05"."X16-1.ANODE MAIN P&P1 ROTARY CCW", signal07 := "BK05"."X17-1.ANODE MAIN P&P1 PRESSURE SWITCH", signal08 := "BK05"."X10-2.ANODE MAIN P&P1 Z-AXIS HOME SENSOR", signal09 := "BK05"."X11-2.SPARE", signal10 := "BK05"."X12-2.ANODE MAIN P&P1 Y-AXIS HOME SENSOR", signal11 := "BK05"."X13-2.SPARE", signal12 := "BK05"."X14-2.SPARE", signal13 := "BK05"."X15-2.SPARE", signal14 := "BK05"."X16-2.ANODE MAIN P&P1 ROTARY CW", signal15 := "BK05"."X17-2.SPARE", interfaceSignals := #statInterfaceSignalsHmi[8].valueSymbolLeft)
      #instSignals8Right(signal00 :=, signal01 :=, signal02 :=, signal03 :=, signal04 :=, signal05 :=, signal06 :=, signal07 :=, signal08 :=, signal09 :=, signal10 :=, signal11 :=, signal12 :=, signal13 :=, signal14 :=, signal15 :=, interfaceSignals := #statInterfaceSignalsHmi[8].valueSymbolRight)
   END_RUNG
   // the same network as SCL:
   #instSignals8Left(signal00 := "BK05"."X10-1.ANODE MAIN P&P1 Z-AXIS LIMIT SENSOR(-)",   // "LAF_InterfaceSignalsBool"
                     signal01 := "BK05"."X11-1.ANODE MAIN P&P1 Z-AXIS LIMIT SENSOR(+)",
                     signal02 := "BK05"."X12-1.ANODE MAIN P&P1 Y-AXIS LIMIT SENSOR(-)",
                     signal03 := "BK05"."X13-1.ANODE MAIN P&P1 Y-AXIS LIMIT SENSOR(+)",
                     signal04 := "BK05"."X14-1.SPARE",
                     signal05 := "BK05"."X15-1.ANODE MAIN P&P1 DETECT SENSOR",
                     signal06 := "BK05"."X16-1.ANODE MAIN P&P1 ROTARY CCW",
                     signal07 := "BK05"."X17-1.ANODE MAIN P&P1 PRESSURE SWITCH",
                     signal08 := "BK05"."X10-2.ANODE MAIN P&P1 Z-AXIS HOME SENSOR",
                     signal09 := "BK05"."X11-2.SPARE",
                     signal10 := "BK05"."X12-2.ANODE MAIN P&P1 Y-AXIS HOME SENSOR",
                     signal11 := "BK05"."X13-2.SPARE",
                     signal12 := "BK05"."X14-2.SPARE",
                     signal13 := "BK05"."X15-2.SPARE",
                     signal14 := "BK05"."X16-2.ANODE MAIN P&P1 ROTARY CW",
                     signal15 := "BK05"."X17-2.SPARE",
                     interfaceSignals := #statInterfaceSignalsHmi[8].valueSymbolLeft,
                     ENO => #_w1);
   IF #_w1 THEN
       #instSignals8Right(interfaceSignals := #statInterfaceSignalsHmi[8].valueSymbolRight);   // "LAF_InterfaceSignalsBool"
   END_IF;
END_REGION

